# B&R Automation Studio project vibratorControlWithCurrentController (part 2)

### Hardware
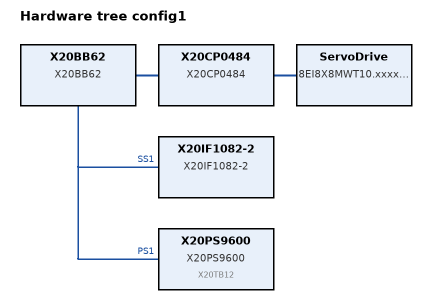
[picture p1: hardware tree config1]
```
ServoDrive : 8EI8X8MWT10.xxxx-1 v2.3.2.0  [PLK1 -> X20CP0484.IF3 (NodeNumber=1) [Cable Type=PowerlinkCable, Length=10, Version=1.0.0.3]]
  MotionTP = Acp10Arnc0
  Ax1Interface = Ax1EnDat
X20BB62 : X20BB62 v1.3.0.0
  Connector IF6:
    CycleTime = 1600
    AsyncPayload = 120
    OutputJustInTime = off
X20CP0484 : X20CP0484 v1.7.0.0  [SL -> X20BB62.SL1]
  Connector IF2:
    ActivateDevice = 1
    HostName = countingmachine
    Mode = Manual
    InternetAddress = 192.168.2.11
    SubnetMask = 255.255.255.0
    InaNodeNumber = 0
    ActivateSnmp = 2
  Connector IF3:
    MtuSize = 1500
    CycleTime = 800
    InternetAddress = 192.168.200.240
    SubnetMask = 255.255.255.0
    ActivateANSL = 1
  ConfigurationID = vibratorControlWithCurrentController
  UserPartitionSize = 100
  RemanentGlobalPvSize = 500
  VolatileGlobalPvSize = 455350
  EnableUsbRemoteInstall = 1
  EnableCfRemoteInstall = 1
  TimerDeviceType = EPLX2X
  TimerDevice = X20CP0484.IF3
  IdleTaskClass = 4
  TaskClassIdleTime = 1600
  CyclicTaskClassCount = 5
  Cyclic1Duration = 800
  Cyclic1Tolerance = 0
  Cyclic2Duration = 1600
  Cyclic2Tolerance = 0
  Cyclic3Duration = 4800
  Cyclic3Tolerance = 0
  Cyclic4Duration = 20000
  Cyclic4Tolerance = 1000000
  Cyclic5Duration = 40000
  Cyclic5Tolerance = 1000000
  Cyclic6Duration = 500000
  Cyclic6Tolerance = 500000
  Cyclic7Duration = 1000000
  Cyclic7Tolerance = 1000000
  Cyclic8Duration = 9600
  Cyclic8Tolerance = 30000000
  FileDevice1
  FileDeviceName1 = USER
  FileDevicePath1 = USER_PATH
  TimeZone = 140
  ActivateSntp = 1
  SntpcServAddr1 = 192.168.1.199
  EthernetHostName = cm20
  EthernetDefaultGateway = 192.168.1.254
  ActivateDns = 1
  DnsServer1 = 192.168.1.1
  FtpUser1
  FtpUsername1 = admin
  FtpUserPassword1 = /xeWp7dP4cZARaoRUYb4lC4ZD6ydIPKFJHxZK63t4D4=
  FtpUserSalt1 = z+XtgaLv
  FTPAccessRight1 = 0
  FtpUser2
  FtpUsername2 = superuser
  FtpUserPassword2 = hun78AKmVJbSvtD9VGxdA3Iq+bPiFMAeRRsTULM9hlc=
  FtpUserSalt2 = IDYkuK0C
  FTPAccessRight2 = 0
  FTPdevice2 = ALL
  FtpUser3
  FtpUsername3 = update
  FtpUserPassword3 = +43P0CP5LPvLZS5Hk18lIwvQq9JpaLJM6nsEQnrbHXY=
  FtpUserSalt3 = TaVVG8PK
  FTPAccessRight3 = 0
  FTPMSpath3 = update
  FtpUser4
  FtpUsername4 = updateewu
  FtpUserPassword4 = epKGN9X0JvLfxgCXyMdS0yy+jyVnLXtvgYSXuK2LydA=  // updateewu
  FtpUserSalt4 = ShQX0Ew+
  FTPAccessRight4 = 0
  FTPMSpath4 = updateewu
  ActivateOpcUa = 1
  OpcUaInformationModels_PV_Version = 2
  OpcUaInformationModel_Facet = 0
  OpcUaInformationModel_TypeInformation = 0
  OpcUaInformationModel_BaseObjectTypeForStructures = 0
X20IF1082-2 : X20IF1082-2 v1.15.0.0  [SS -> X20BB62.SS1]
  Connector IF1:
    Operation = EthOnly
    HostName = cm20
    ActivateANSL = 1
    ActivateSnmp = 2
X20PS9600 : X20PS9600 v1.6.1.0  [PS -> X20BB62.PS1; SS1 -> X20TB12.SS]
X20TB12 : X20TB12 v1.0.0.0
```

### Acp10map.ncm - X20CP0484/Motion/Acp10map.ncm
```
NcMapping (NcSwId=Acp10, DisabledNodesAreHidden=False)
  NcObject gAxisBelt (ModuleId=ServoDrive, Type=ncAXIS, Channel=1, AcoposSimulation=Off, InitParameter=gAxisBelti, AcoposParameter=gAxisBelta, Disabled=TRUE, ModuleDisabled=FALSE)
  NcObject gAxisVibL (ModuleId=ServoDrive, Type=ncAXIS, Channel=2, AcoposSimulation=Off, InitParameter=gAxisVibLi, AcoposParameter=lfNew, Disabled=TRUE, ModuleDisabled=FALSE)
  NcObject 8EI8X8MWT10.xxxx-1_ncV_AXIS1 (ModuleId=ServoDrive, Type=ncV_AXIS, Channel=1, Disabled=TRUE, ModuleDisabled=FALSE)
  NcObject 8EI8X8MWT10.xxxx-1_ncV_AXIS2 (ModuleId=ServoDrive, Type=ncV_AXIS, Channel=2, Disabled=TRUE, ModuleDisabled=FALSE)
  NcObject gAxisVibC (ModuleId=ServoDrive, Type=ncAXIS, Channel=3, AcoposSimulation=Off, InitParameter=gAxisVibCi, AcoposParameter=cfCurCtr, Disabled=FALSE, ModuleDisabled=FALSE)
  NcObject ServoDrive_ncV_AXIS3 (ModuleId=ServoDrive, Type=ncV_AXIS, Channel=3, AcoposSimulation=off, Disabled=true, ModuleDisabled=FALSE)
```

## Logical view

Binary libraries used (declarations not repeated): operator, runtime, astime, AsIecCon, Acp10man, Acp10par, NcGlobal, MpRecipe, MpBase, sys_lib, MpAlarmX, Acp10_MC, AsBrMath, standard, AsBrStr, brsystem, DataObj, AsOpcUas, ArProject, AsSem, AsIO, AsOpcUac, FileIO, AsIODiag, AsUSB, RandomLib, AsHttp, AsARCfg, AsMath, asstring, AsEthIP, MTTypes, MpData, MpServer, EasyUaClnt, AsIOLink, AsIOAcc, AsUDP, MTData, MTBasics, MTFilter, MTLookUp 5.24.1, MpReport 5.23.1

### Global.typ - Global data types
```iecst
TYPE
	copy_recipe_command_typ :
		(
		COPY_RECIPE_NONE := 0,
		COPY_RECIPE_NEXT_TO_WORKING := 1,
		COPY_RECIPE_SANDBOX_TO_NEXT := 2
		);
END_TYPE
```

### Global.var - Global variables
```iecst
VAR
	gMachineType : STRING[10];
END_VAR
VAR CONSTANT
	MODE_EMPTY : DINT := 21;
	MODE_TEACH_CAPCON : DINT := 25;
	MODE_TEACH_BELT : DINT := 26;
END_VAR
VAR
	gAxisVibC : ACP10AXIS_typ;
	gAxisVibL : ACP10AXIS_typ;
	gAxisBelt : ACP10AXIS_typ;
END_VAR
```

### Package Logical/Libraries - Global libraries

### Library Logical/Libraries/brdkMC (IEC, version 2.02.2) - Basic motion library
Depends on: Runtime, Acp10_MC, AsBrMath, standard, AsBrStr

#### brdkMC.typ - Exported data types
```iecst
TYPE
	brdk_mc_para_hwinputs_typ : 	STRUCT  (*HW inputs*)
		homeReference : brdk_mc_para_hwinputs_di_typ; (*Home switch*)
		negHwLimit : brdk_mc_para_hwinputs_di_typ; (*Negative hw limit switch*)
		posHwLimit : brdk_mc_para_hwinputs_di_typ; (*Positive hw limit switch*)
		trigger1 : brdk_mc_para_hwinputs_di_typ; (*Trigger switch*)
		trigger2 : brdk_mc_para_hwinputs_di_typ; (*Trigger switch*)
	END_STRUCT;
	brdk_mc_para_hwinputs_di_typ : 	STRUCT  (*HW input commands*)
		input : BOOL; (*Manipulates switch in the drive if useExternalInput is TRUE*)
		useExternalInput : BOOL; (*Get the input from a digital input module or PLC*)
	END_STRUCT;
	brdk_mc_command_typ : 	STRUCT  (*Commands*)
		power : BOOL; (*Power on drive*)
		home : BOOL; (*Home axis*)
		moveAbsolute : BOOL; (*Move to position*)
		moveAdditive : BOOL; (*Move distance*)
		moveVelocity : BOOL; (*Move with speed*)
		halt : BOOL; (*Halt movement*)
		stop : BOOL; (*Stop movement*)
		jogPositive : BOOL; (*Jog in positive direction*)
		jogNegative : BOOL; (*Jog in negative direction*)
		gearIn : BOOL; (*Connect slave axis to master axis*)
		gearOut : BOOL; (*Disconnect master and slave axes*)
		limitLoad : BOOL; (*Limits the motor torque*)
		errorAcknowledge : BOOL; (*Acknowledge error at rising edge*)
		updatePeriod : BOOL; (*Update axis factor and period, done automatically at axis bootup*)
		simulateError : BOOL; (*Trigger a simulated axis error*)
		resetTorqueStatus : BOOL; (*Reset torque statistics*)
		newBatAcknowledge : BOOL; (*Acknowledge battery excange - Only for AcoposMicro with Endat 2.2*)
	END_STRUCT;
	brdk_mc_status_typ : 	STRUCT  (*Status*)
		state : Status_enum; (*Current PLCopen state*)
		actVelocity : REAL; (*Actual velocity [PLCopen units/s]*)
		actPosition : REAL; (*Actual position [PLCopen units]*)
		actLagError : REAL; (*Actual position lag error [PLCopen units] if configuration factor set > 0 else in [units]*)
		actTorque : REAL; (*Actual torque [Nm]*)
		torque : brdk_mc_status_torque_typ; (*Extended torque readout*)
		powerOn : BOOL; (*Axis is powered on*)
		isHomed : BOOL; (*Axis is homed*)
		inMotion : BOOL; (*Axis is in motion or geared in to a master axis*)
		stopped : BOOL; (*Axis is stopped using the command stop and is at standstill*)
		done : BOOL; (*Specified command done*)
		busy : BOOL; (*Specified command is executed and active*)
		updateDone : BOOL; (*UpdatePeriod command done*)
		error : brdk_mc_status_error_typ; (*Error status information*)
		driveStatus : brdk_mc_status_drive_status_typ; (*Drive status information*)
		encoderBatteryStatus : brdk_mc_enc_bat_status_typ; (*Status of encoder battery - Only for AcoposMicro with Endat 2.2*)
		axisDescription : STRING[30]; (*Defined axis desciption*)
	END_STRUCT;
	brdk_mc_status_drive_status_typ : 	STRUCT  (*Drive status*)
		simulation : BOOL; (*If TRUE, simulation mode is active for the drive.*)
		initialized : BOOL; (*If TRUE, the network is initialized.*)
		homeSwitch : BOOL; (*If TRUE, the digital reference switch input is active.*)
		posLimitSwitch : BOOL; (*If TRUE, the positive hardware limit switch is active.*)
		negLimitSwitch : BOOL; (*If TRUE, the negative hardware limit switch is active.*)
		trigger1 : BOOL; (*If TRUE, the first trigger input is active.*)
		trigger2 : BOOL; (*If TRUE, the second trigger input is active.*)
		driveEnable : BOOL; (*If TRUE, the enable input is in use.*)
		controllerReady : BOOL; (*If TRUE, the controller is ready to be turned on.*)
		lagWarning : BOOL; (*If TRUE, the lag error has exceeded the limit value specified for a warning (limit.parameter.ds_warning).*)
	END_STRUCT;
	brdk_mc_status_error_text_typ : 	STRUCT  (*Error text*)
		active : ARRAY[0..4]OF STRING[363]; (*Active fault descriptions*)
		last : ARRAY[0..4]OF STRING[363]; (*Last reset faults descriptions*)
	END_STRUCT;
	brdk_mc_status_error_typ : 	STRUCT  (*Error status*)
		fault : BOOL; (*Fault present on axis*)
		count : UINT; (*Number of faults*)
		text : brdk_mc_status_error_text_typ; (*Error message*)
	END_STRUCT;
	brdk_mc_status_torque_typ : 	STRUCT  (*Torque status*)
		actual : REAL; (*Actual torque 0.5 sec average [Nm]*)
		continous : REAL; (*Continous peak torque 5 sec average [Nm]*)
		peak : REAL; (*Peak torque 0.5 sec average [Nm]*)
	END_STRUCT;
	brdk_mc_internal_typ : 	STRUCT  (*internal*)
		MC_BR_CyclicRead_1 : MC_BR_CyclicRead;
		MC_MoveVelocity_0 : MC_MoveVelocity;
		MC_Reset_0 : MC_Reset;
		MC_Home_0 : MC_Home;
		MC_Halt_0 : MC_Halt;
		MC_Stop_0 : MC_Stop;
		MC_Power_0 : MC_Power;
		MC_BR_Simulation_0 : MC_BR_Simulation;
		MC_ReadActualPosition_0 : MC_ReadActualPosition;
		MC_ReadStatus_0 : MC_ReadStatus;
		MC_ReadActualVelocity_0 : MC_ReadActualVelocity;
		MC_GearIn_0 : MC_GearIn;
		MC_GearOut_0 : MC_GearOut;
		MC_MoveAdditive_0 : MC_MoveAdditive;
		MC_MoveAbsolute_0 : MC_MoveAbsolute;
		MC_ReadActualTorque_0 : MC_ReadActualTorque;
		MC_BR_ReadDriveStatus_0 : MC_BR_ReadDriveStatus;
		MC_BR_ReadAxisError_0 : MC_BR_ReadAxisError;
		MC_BR_AxisErrorCollector_0 : MC_BR_AxisErrorCollector;
		MC_BR_GetHardwareInfo_0 : MC_BR_GetHardwareInfo;
		MC_BR_SetHardwareInputs_0 : MC_BR_SetHardwareInputs;
		MC_BR_InitAxisSubjectPar_0 : MC_BR_InitAxisSubjectPar;
		MC_BR_CyclicRead_0 : MC_BR_CyclicRead;
		MC_BR_ReadParID_3 : MC_BR_ReadParID;
		MC_BR_ReadParID_2 : MC_BR_ReadParID;
		MC_BR_ReadParID_1 : MC_BR_ReadParID;
		MC_BR_ReadParID_0 : MC_BR_ReadParID;
		MC_BR_InitModPos_0 : MC_BR_InitModPos;
		MC_BR_CommandError_0 : MC_BR_CommandError;
		MC_BR_WriteParID_1 : MC_BR_WriteParID;
		MC_BR_WriteParID_0 : MC_BR_WriteParID;
		MC_LimitLoad_0 : MC_LimitLoad;
		encoderReset : UDINT;
		old_hardwareInput : brdk_mc_para_hwinputs_typ;
		encoderStatus : UDINT;
		encoderType : USINT;
		strcat_adr : UDINT;
		string2 : STRING[8];
		tmpErrorString : STRING[324];
		tmpErrorCount : UINT;
		tmpErrorID : STRING[5];
		tmpErrorArray : ARRAY[0..3]OF STRING[80];
		i : USINT;
		oldParID : UINT;
		oldErrorID : UINT;
		substate : USINT;
		tmpNumberOfErrors : UINT;
		filterBase : ARRAY[0..1]OF REAL;
		RTInfo : RTInfo;
		calcActualValueTemp_old : REAL;
		calcActualValueTemp : REAL;
		calcActualValue_old : ARRAY[0..1]OF REAL;
		calcActualValue : ARRAY[0..1]OF REAL;
		filterTime : ARRAY[0..1]OF REAL;
		stateMotor : USINT;
		filterBaseTemp : REAL;
		filterTimeTemp : REAL;
		TON_error_read_delay : TON;
		k : USINT;
		batteryState : bat_state_enum;
		acoposMicroBatMon : BOOL;
		tmpDriveStatus : MC_DRIVESTATUS_TYP;
		initialized : BOOL;
	END_STRUCT;
	brdk_mc_parameter_typ : 	STRUCT  (*Parameters*)
		position : REAL; (*Position for an absolute movement [PLCopen units]*)
		distance : REAL; (*Distance for an additive movement [PLCopen units]*)
		velocity : REAL; (*Movement velocity [PLCopen units/s] *)
		acceleration : REAL; (*Acceleration [PLCopen units/s²]*)
		deceleration : REAL; (*Deceleration [PLCopen units/s²]*)
		decelerationFault : REAL; (*Deceleration at axis fault [PLCopen units/s²]*)
		direction : USINT; (*Movement direction:
mcPOSITITVE_DIR ... 0

mcNEGATIVE_DIR ... 1

mcCURRENT_DIR ... 2

mcSHORTEST_WAY ... 3

mcEXCEED_PERIOD ... 8*)
		loadLimit : REAL; (*Torque load limit [Nm]*)
		homePosition : REAL; (*Home position, position after homing [PLCopen units]*)
		homeMode : USINT; (*Homing mode:
mcHOME_ABS_SWITCH (performs homing with absolute reference switch)

mcHOME_SWITCH_GATE (homing with reference switch gate)

mcHOME_LIMIT_SWITCH (homing with hardware limit switch)

mcHOME_DIRECT (direct homing without reference pulse)

mcHOME_REF_PULSE (direct homing with reference pulse)

mcHOME_ABSOLUTE (homing by setting the homing offset)

mcHOME_ABSOLUTE_CORR (homing by setting the homing offset with counting range correction)

mcHOME_DCM (homing using interval-encoded reference marks)

mcHOME_DCM_CORR (Homing using distance coded reference marks with counting range correction)

mcHOME_RESTORE_POS (restore position from permanent memory)

mcHOME_AXIS_REF (performs homing with the data from the axis structure)

mcHOME_BLOCK_TORQUE (performs homing to mechanical limit, torque as criteria)

mcHOME_BLOCK_DS (performs homing to mechanical limit, lag error value as criteria)*)
		ratioSlave : INT; (*Slave gear ratio*)
		ratioMaster : UINT; (*Master gear ration*)
		gearInMasterParID : UINT; (*This ParID is used instead of the position setpoint;
0 ... Use position setpoint*)
		gearInMasterParIDMaxVelocity : REAL; (*If this parameter is "0.0", the current velocity of the master axis is used.
If a value is specified for "MasterParID":
Maximum velocity of the master ParID value

If a value is not specified for "MasterParID":
Maximum velocity of the master axis [PLCopen units of master/s]*)
		errorSimulationCommand : USINT; (*0: Warning message reported

1: Error message reported

2: Error message reported and active movement aborted

3: Error message reported, active movement aborted and controller switched off

4: Error message reported, active movement ended with a speed-controlled ramp and controller switched off*)
		hwInput : brdk_mc_para_hwinputs_typ; (*Hardware input manipulation for home reference, triggers and limit switches*)
	END_STRUCT;
	brdk_mc_configuration_typ : 	STRUCT  (*Axis configuration*)
		masterAxis : UDINT; (*Master axis reference*)
		axis : UDINT; (*Axis reference*)
		errorTextObject : STRING[12]; (*Name of the acp10 error text object
If no name is entered, the default name 'acp10etxen' is assumed (table must be available in the project)*)
		description : STRING[30]; (*Optional: Axis description or name; added to the error texts*)
		factor : UDINT; (*Axis factor*)
		period : UDINT; (*Axis period*)
		ignoreSwLimit : USINT; (*Ignore software end limit positions (0: end limits active 1: ignore sw end limits)*)
		disableVelocityReading : BOOL; (*Disables actual velocity status readout*)
		disablePositionReading : BOOL; (*Disables actual position status readout*)
		disableTorqueReading : BOOL; (*Disables actual torque status readout*)
		disableTemperatureReading : BOOL; (*Disables actual motor temperature readout*)
		disableLagErrorReading : BOOL; (*Disables actual lag error status readout*)
	END_STRUCT;
	brdk_mc_info_typ : 	STRUCT  (*HW info*)
		startupPhase : STRING[100]; (*Drive startup phase information*)
		hw : brdk_mc_info_hw_typ; (*Hardware information*)
	END_STRUCT;
	brdk_mc_info_hw_typ : 	STRUCT  (*Hardware information*)
		drive : brdk_mc_info_hw_drive_typ; (*Motor type*)
		motor : brdk_mc_info_hw_motor_typ; (*Motors maximum torque [Nm]*)
	END_STRUCT;
	brdk_mc_info_hw_drive_typ : 	STRUCT  (*HW drive info*)
		model : STRING[32]; (*Drive model number*)
		serial : STRING[32]; (*Drive serial number*)
		card : ARRAY[0..3]OF brdk_mc_info_hw_card_typ; (*Plugin cards*)
	END_STRUCT;
	brdk_mc_info_hw_card_typ : 	STRUCT  (*HW card info*)
		model : STRING[32]; (*Model number*)
		serial : STRING[32]; (*Serial number*)
	END_STRUCT;
	brdk_mc_info_hw_motor_typ : 	STRUCT  (*Motor info*)
		model : STRING[32]; (*Motor type*)
		temperature : REAL; (*Motor temperature [C]*)
		torqueRated : REAL; (*Motors nominal torque [Nm]*)
		torqueMaximum : REAL; (*Motors maximum torque [Nm]*)
	END_STRUCT;
	brdk_mc_enc_bat_status_typ : 	STRUCT  (*Encoder battry information*)
		batteryOK : BOOL; (*Encoder battery is OK - Voltage OK and position valid*)
		batteryError : BOOL; (*Encoder battery NOT ok - voltage has dropped below threshhold. Posiion valid if PositionLost = false.*)
		batteryWarning : BOOL; (*Error has been acknowledged - battery not exchanged, position still valid*)
		positionLost : BOOL; (*Encoder postion has been lost due to battery failure*)
	END_STRUCT;
	state_enum :
		(
		ST_INIT := 0,
		ST_WAIT := 1,
		ST_POWER_ON := 2,
		ST_HOME_AT_POWER_OFF := 3,
		ST_EXTERNAL_HW_INPUTS := 5,
		ST_UPDATE_FACTOR_PERIOD := 6,
		ST_READY := 10,
		ST_HOME := 20,
		ST_STOP := 30,
		ST_HALT := 31,
		ST_MOVE_ABSOLUTE := 40,
		ST_MOVE_ADDITIVE := 41,
		ST_MOVE_VELOCITY := 42,
		ST_GEAR_START := 50,
		ST_GEAR_STOP := 51,
		ST_IN_GEAR := 52,
		ST_JOG_POS := 60,
		ST_JOG_NEG := 61,
		ST_HALT_JOG := 62,
		ST_STOP_AFTER_ERROR := 100,
		ST_STOPPING_AFTER_ERROR := 101,
		ST_ERROR := 110,
		ST_CHECK_ERROR := 111,
		ST_ERROR_RESET := 120,
		ST_ENCODER_ERROR_RESET := 130
		);
	bat_state_enum :
		(
		ST_BAT_OK := 0,
		ST_BAT_ERROR := 1,
		ST_BAT_WARNING := 2,
		ST_BAT_POS_LOST := 3
		);
	Status_enum :
		(
		DISABLED := 0,
		STANDSTILL := 1,
		HOMING := 2,
		CONTINOUS_MOTION := 3,
		DISCRETE_MOTION := 4,
		SYNCHRONIZED_MOTION := 5,
		STOPPING := 6,
		ERROR_STOP := 10
		);
END_TYPE
```

#### brdkMC.fun - Exported functions and function blocks
```iecst
FUNCTION_BLOCK brdkMcBasic (*brdk Motion basic*)
	VAR_INPUT
		command : brdk_mc_command_typ; (*command input*)
		parameter : brdk_mc_parameter_typ; (*parameter input*)
		configuration : brdk_mc_configuration_typ; (*configuration input*)
	END_VAR
	VAR_OUTPUT
		status : brdk_mc_status_typ; (*status output*)
		info : brdk_mc_info_typ; (*information output*)
	END_VAR
	VAR
		state : state_enum; (*state enumeration*)
		internal : brdk_mc_internal_typ; (*internal structure*)
		pAxis : REFERENCE TO ACP10AXIS_typ; (*internal axis pointer reference*)
	END_VAR
END_FUNCTION_BLOCK

FUNCTION dstoa : UINT (****)
	VAR_INPUT
		driveState : Status_enum;
		pString : UDINT;
	END_VAR
END_FUNCTION
```

#### brdkMcBasic.st
```iecst
FUNCTION_BLOCK  brdkMcBasic

	(* Access the axis structure *)
	pAxis ACCESS configuration.axis;

	(*********************** CHECK FOR ERRORS **************************)
	IF (state < ST_STOP_AFTER_ERROR) THEN
		IF (internal.MC_BR_AxisErrorCollector_0.Errorstop) THEN
			state := ST_ERROR;
		ELSIF (internal.MC_BR_AxisErrorCollector_0.FunctionBlockError) OR
		   	  (internal.MC_BR_AxisErrorCollector_0.AxisError) OR
			  (internal.MC_BR_AxisErrorCollector_0.AxisWarning) THEN
			status.busy := 0;
			status.done := 0;
			state 		:= ST_STOP_AFTER_ERROR;
		END_IF
	END_IF

	(***************** CHECK IF POWER SHOULD BE OFF *******************)
	IF (command.power = 0 AND state < ST_STOP_AFTER_ERROR AND state <> ST_HOME_AT_POWER_OFF AND state <> ST_INIT AND state <> ST_EXTERNAL_HW_INPUTS AND state <> ST_UPDATE_FACTOR_PERIOD) THEN
		status.busy := 0;
		status.done := 0;

		IF ((internal.MC_ReadStatus_0.Errorstop = 1) AND (internal.MC_ReadStatus_0.Valid = TRUE)) THEN
			state := ST_ERROR_RESET;
		ELSE
			state := ST_WAIT;
		END_IF
	END_IF

	(* Status Motion States *)
	IF internal.MC_ReadStatus_0.Disabled THEN
		status.state := DISABLED;
	ELSIF internal.MC_ReadStatus_0.StandStill THEN
		status.state := STANDSTILL;
	ELSIF internal.MC_ReadStatus_0.Homing THEN
		status.state := HOMING;
	ELSIF internal.MC_ReadStatus_0.Stopping THEN
		status.state := STOPPING;
	ELSIF internal.MC_ReadStatus_0.Errorstop THEN
		status.state := ERROR_STOP;
	ELSIF internal.MC_ReadStatus_0.DiscreteMotion THEN
		status.state := DISCRETE_MOTION;
	ELSIF internal.MC_ReadStatus_0.ContinuousMotion THEN
		status.state := CONTINOUS_MOTION;
	ELSIF internal.MC_ReadStatus_0.SynchronizedMotion THEN
		status.state := SYNCHRONIZED_MOTION;
	END_IF

	(* Limit load torque *)
	internal.MC_LimitLoad_0.Load		:= parameter.loadLimit;
	internal.MC_LimitLoad_0.Direction	:= parameter.direction;
	internal.MC_LimitLoad_0.Enable		:= command.limitLoad;

	(***************************************************************)
	(************************* MAIN CONTROL ************************)
	(***************************************************************)

	(* check for stop command *)
	IF command.stop AND state <> ST_INIT AND state <> ST_WAIT AND state <> ST_POWER_ON AND state <> ST_UPDATE_FACTOR_PERIOD AND state <> ST_HOME_AT_POWER_OFF AND state <> ST_EXTERNAL_HW_INPUTS AND state <> ST_STOP AND state < 100 THEN
		internal.MC_Stop_0.Deceleration	:= parameter.deceleration;
		internal.MC_Stop_0.Execute 		:= 1;
		state := ST_STOP;
	END_IF

	CASE state OF

		(****************** STARTING DRIVE *****************)
		ST_INIT:
			CASE internal.substate OF
				0:
					IF pAxis.network.phase = 90 THEN
						internal.substate := 10;
					END_IF

				10:	(* initialize factor and period *)
					internal.MC_BR_InitModPos_0.Factor	:= configuration.factor;
					internal.MC_BR_InitModPos_0.Period	:= configuration.period;
					internal.MC_BR_InitModPos_0.Execute	:= TRUE;

					IF internal.MC_BR_InitModPos_0.Done THEN
						internal.MC_BR_InitModPos_0.Execute := FALSE;
						internal.substate					:= 20;
					END_IF

				20: (* set end limit ignore *)
					internal.MC_BR_WriteParID_1.ParID		:= ACP10PAR_SGEN_SW_END_IGNORE;
					internal.MC_BR_WriteParID_1.DataType	:= ncPAR_TYP_USINT;
					internal.MC_BR_WriteParID_1.DataAddress	:= ADR(configuration.ignoreSwLimit);
					internal.MC_BR_WriteParID_1.Execute		:= TRUE;

					IF internal.MC_BR_WriteParID_1.Done THEN
						internal.MC_BR_WriteParID_1.Execute := FALSE;
						internal.initialized				:= TRUE;
						internal.substate 					:= 0;
						state 								:= ST_WAIT;
					END_IF
					internal.MC_BR_WriteParID_1(Axis := configuration.axis);
			END_CASE

		(******************** WAIT *************************)
		ST_WAIT: (* STATE: Wait *)

			(* reset status *)
			status.busy   		:= 0;
			status.done 		:= 0;
			status.updateDone 	:= 0;

			(* reset user commands *)
			command.stop 			:= 0;
			command.halt 			:= 0;
			command.moveVelocity	:= 0;
			command.moveAbsolute	:= 0;
			command.moveAdditive	:= 0;
			command.gearIn 			:= 0;
			command.gearOut			:= 0;
			command.jogPositive		:= 0;
			command.jogNegative		:= 0;

			(* reset all fb execute inputs we use *)
			internal.MC_Home_0.Execute 					:= 0;
			internal.MC_Stop_0.Execute 					:= 0;
			internal.MC_Halt_0.Execute 					:= 0;
			internal.MC_MoveAbsolute_0.Execute 			:= 0;
			internal.MC_MoveAdditive_0.Execute 			:= 0;
			internal.MC_MoveVelocity_0.Execute 			:= 0;
			internal.MC_GearIn_0.Execute 				:= 0;
			internal.MC_GearOut_0.Execute 				:= 0;
			internal.MC_BR_ReadAxisError_0.Acknowledge	:= 0;
			internal.MC_Reset_0.Execute 				:= 0;
			internal.substate 							:= 0;

			IF (command.power) THEN
				state := ST_POWER_ON;
			ELSE
				internal.MC_Power_0.Enable := 0;
			END_IF

			(* wait for homing command *)
			IF (command.home) THEN
				internal.MC_Home_0.Position 	:= parameter.homePosition;
				internal.MC_Home_0.HomingMode 	:= parameter.homeMode;
				internal.MC_Home_0.Execute 		:= 1;
				state 							:= ST_HOME_AT_POWER_OFF;
			END_IF

			(* initialize factor and period *)
			IF command.updatePeriod THEN
				internal.MC_BR_InitModPos_0.Axis 	:= configuration.axis;
				internal.MC_BR_InitModPos_0.Factor	:= configuration.factor;
				internal.MC_BR_InitModPos_0.Period	:= configuration.period;
				internal.MC_BR_InitModPos_0.Execute	:= TRUE;
				state 								:= ST_UPDATE_FACTOR_PERIOD;
			END_IF

			(* check if external inputs has been changed *)
			IF parameter.hwInput.homeReference.useExternalInput <> internal.old_hardwareInput.homeReference.useExternalInput OR
			   parameter.hwInput.negHwLimit.useExternalInput <> internal.old_hardwareInput.negHwLimit.useExternalInput OR
			   parameter.hwInput.posHwLimit.useExternalInput <> internal.old_hardwareInput.posHwLimit.useExternalInput OR
			   parameter.hwInput.trigger1.useExternalInput <> internal.old_hardwareInput.trigger1.useExternalInput OR
			   parameter.hwInput.trigger2.useExternalInput <> internal.old_hardwareInput.trigger2.useExternalInput THEN
				IF parameter.hwInput.homeReference.useExternalInput <> internal.old_hardwareInput.homeReference.useExternalInput THEN
					IF parameter.hwInput.homeReference.useExternalInput THEN
						pAxis.dig_in.level.reference.5 := pAxis.dig_in.level.reference.8 := 1;
					ELSE
						pAxis.dig_in.level.reference.5 := pAxis.dig_in.level.reference.8 := 0;
					END_IF
				END_IF
				IF parameter.hwInput.negHwLimit.useExternalInput <> internal.old_hardwareInput.negHwLimit.useExternalInput THEN
					IF parameter.hwInput.negHwLimit.useExternalInput THEN
						pAxis.dig_in.level.neg_hw_end.5 := pAxis.dig_in.level.neg_hw_end.8 := 1;
					ELSE
						pAxis.dig_in.level.neg_hw_end.5 := pAxis.dig_in.level.neg_hw_end.8 := 0;
					END_IF
				END_IF
				IF parameter.hwInput.posHwLimit.useExternalInput <> internal.old_hardwareInput.posHwLimit.useExternalInput THEN
					IF parameter.hwInput.posHwLimit.useExternalInput THEN
						pAxis.dig_in.level.pos_hw_end.5 := pAxis.dig_in.level.pos_hw_end.8 := 1;
					ELSE
						pAxis.dig_in.level.pos_hw_end.5 := pAxis.dig_in.level.pos_hw_end.8 := 0;
					END_IF
				END_IF
				IF parameter.hwInput.trigger1.useExternalInput <> internal.old_hardwareInput.trigger1.useExternalInput THEN
					IF parameter.hwInput.trigger1.useExternalInput THEN
						pAxis.dig_in.level.trigger1.5 := pAxis.dig_in.level.trigger1.8 := 1;
					ELSE
						pAxis.dig_in.level.trigger1.5 := pAxis.dig_in.level.trigger1.8 := 0;
					END_IF
				END_IF
				IF parameter.hwInput.trigger2.useExternalInput <> internal.old_hardwareInput.trigger2.useExternalInput THEN
					IF parameter.hwInput.trigger2.useExternalInput THEN
						pAxis.dig_in.level.trigger2.5 := pAxis.dig_in.level.trigger2.8 := 1;
					ELSE
						pAxis.dig_in.level.trigger2.5 := pAxis.dig_in.level.trigger2.8 := 0;
					END_IF
				END_IF

				internal.old_hardwareInput.homeReference.useExternalInput 	:= parameter.hwInput.homeReference.useExternalInput;
				internal.old_hardwareInput.negHwLimit.useExternalInput 		:= parameter.hwInput.negHwLimit.useExternalInput;
				internal.old_hardwareInput.posHwLimit.useExternalInput 		:= parameter.hwInput.posHwLimit.useExternalInput;
				internal.old_hardwareInput.trigger1.useExternalInput 		:= parameter.hwInput.trigger1.useExternalInput;
				internal.old_hardwareInput.trigger2.useExternalInput 		:= parameter.hwInput.trigger2.useExternalInput;
				state 														:= ST_EXTERNAL_HW_INPUTS;
			END_IF

			(* check if drive was initialized *)
			IF NOT internal.initialized	THEN
				internal.substate := 0;
				state 			  := ST_INIT;
			END_IF

		(******************** POWER ON **********************)
		ST_POWER_ON: (* STATE: Power on *)
			internal.MC_Power_0.Enable := 1;
			IF (internal.MC_Power_0.Status = 1) THEN
				state := ST_READY;
			END_IF

			(* check if error occured *)
			IF (internal.MC_Power_0.Error) THEN
				internal.MC_Power_0.Enable := 0;
				state := ST_WAIT;
			END_IF

		(******************** HOME AT POWER OFF *************)
		ST_HOME_AT_POWER_OFF: (* STATE: start homing process *)
			(* check if functionblock is busy *)
			status.busy := internal.MC_Home_0.Busy;

			(* if axis homed go to state ready *)
			status.done := internal.MC_Home_0.Done;

			(* return to ready state *)
			IF NOT command.home THEN
				status.busy := 0;
				status.done := 0;
				internal.MC_Home_0.Execute := 0;
				state := ST_WAIT;
			END_IF

		(********* setup EXTERNAL HW INPUTS **************)
		ST_EXTERNAL_HW_INPUTS:
			(* check if functionblock is busy *)
			status.busy := internal.MC_BR_InitAxisSubjectPar_0.Busy;

			(* check if command is done *)
			status.done := internal.MC_BR_InitAxisSubjectPar_0.Done;

			internal.MC_BR_InitAxisSubjectPar_0.Execute := TRUE;

			IF internal.MC_BR_InitAxisSubjectPar_0.Done THEN
				internal.MC_BR_InitAxisSubjectPar_0.Execute := FALSE;
				state 										:= ST_WAIT;
			END_IF

		(********* UPDATE period AND factor **************)
		ST_UPDATE_FACTOR_PERIOD:
			status.updateDone := internal.MC_BR_InitModPos_0.Done AND internal.MC_BR_WriteParID_1.Done;

			IF internal.MC_BR_InitModPos_0.Done THEN
				internal.MC_BR_WriteParID_1.ParID		:= ACP10PAR_SGEN_SW_END_IGNORE;
				internal.MC_BR_WriteParID_1.DataType	:= ncPAR_TYP_USINT;
				internal.MC_BR_WriteParID_1.DataAddress	:= ADR(configuration.ignoreSwLimit);
				internal.MC_BR_WriteParID_1.Execute		:= TRUE;
			END_IF

			IF NOT command.updatePeriod THEN
				internal.MC_BR_WriteParID_1.Execute	:= FALSE;
				internal.MC_BR_InitModPos_0.Execute := FALSE;
				state 	 							:= ST_WAIT;
			END_IF

		(******************** READY **********************)
		ST_READY: (* STATE: Waiting for commands *)
			IF command.home AND NOT internal.MC_Home_0.CommandAborted THEN
				internal.MC_Home_0.Position 	:= parameter.homePosition;
				internal.MC_Home_0.HomingMode 	:= parameter.homeMode;
				state := ST_HOME;

			ELSIF command.halt AND NOT internal.MC_Halt_0.CommandAborted THEN
				internal.MC_Halt_0.Deceleration	:= parameter.deceleration;
				state := ST_HALT;

			ELSIF command.moveAbsolute AND NOT internal.MC_MoveAbsolute_0.CommandAborted THEN
				internal.MC_MoveAbsolute_0.Position		:= parameter.position;
				internal.MC_MoveAbsolute_0.Velocity		:= parameter.velocity;
				internal.MC_MoveAbsolute_0.Acceleration	:= parameter.acceleration;
				internal.MC_MoveAbsolute_0.Deceleration	:= parameter.deceleration;
				internal.MC_MoveAbsolute_0.Direction	:= parameter.direction;
				state := ST_MOVE_ABSOLUTE;

			ELSIF command.moveAdditive AND NOT internal.MC_MoveAdditive_0.CommandAborted THEN
				internal.MC_MoveAdditive_0.Distance		:= parameter.distance;
				internal.MC_MoveAdditive_0.Velocity		:= parameter.velocity;
				internal.MC_MoveAdditive_0.Acceleration	:= parameter.acceleration;
				internal.MC_MoveAdditive_0.Deceleration	:= parameter.deceleration;
				state := ST_MOVE_ADDITIVE;

			ELSIF command.moveVelocity AND NOT internal.MC_MoveVelocity_0.CommandAborted THEN
				internal.MC_MoveVelocity_0.Velocity		:= parameter.velocity;
				internal.MC_MoveVelocity_0.Acceleration	:= parameter.acceleration;
				internal.MC_MoveVelocity_0.Deceleration	:= parameter.deceleration;
				internal.MC_MoveVelocity_0.Direction	:= parameter.direction;
				state := ST_MOVE_VELOCITY;

			ELSIF command.jogPositive AND NOT internal.MC_MoveVelocity_0.CommandAborted THEN
				internal.MC_MoveVelocity_0.Velocity		:= parameter.velocity;
				internal.MC_MoveVelocity_0.Acceleration	:= parameter.acceleration;
				internal.MC_MoveVelocity_0.Deceleration	:= parameter.deceleration;
				internal.MC_MoveVelocity_0.Direction	:= mcPOSITIVE_DIR;
				state := ST_JOG_POS;

			ELSIF command.jogNegative AND NOT internal.MC_MoveVelocity_0.CommandAborted THEN
				internal.MC_MoveVelocity_0.Velocity		:= parameter.velocity;
				internal.MC_MoveVelocity_0.Acceleration	:= parameter.acceleration;
				internal.MC_MoveVelocity_0.Deceleration	:= parameter.deceleration;
				internal.MC_MoveVelocity_0.Direction	:= mcNEGATIVE_DIR;
				state := ST_JOG_NEG;

			ELSIF command.gearIn AND NOT internal.MC_GearIn_0.CommandAborted THEN
				internal.MC_GearIn_0.RatioNumerator			:= parameter.ratioSlave;
				internal.MC_GearIn_0.RatioDenominator		:= parameter.ratioMaster;
				internal.MC_GearIn_0.Acceleration			:= parameter.acceleration;
				internal.MC_GearIn_0.Deceleration			:= parameter.deceleration;
				internal.MC_GearIn_0.MasterParID 			:= parameter.gearInMasterParID;
				internal.MC_GearIn_0.MasterParIDMaxVelocity := parameter.gearInMasterParIDMaxVelocity;
				state := ST_GEAR_START;
			ELSIF command.gearOut THEN
			 	state := ST_GEAR_STOP;
			END_IF

			status.busy	:= 0;
			status.done := 0;

			internal.MC_Home_0.Execute			:= command.home;
			internal.MC_Halt_0.Execute			:= command.halt;
			internal.MC_MoveVelocity_0.Execute  := command.moveVelocity OR command.jogPositive OR command.jogNegative;
			internal.MC_MoveAbsolute_0.Execute 	:= command.moveAbsolute;
			internal.MC_MoveAdditive_0.Execute 	:= command.moveAdditive;
			internal.MC_GearIn_0.Execute 		:= command.gearIn;
			internal.MC_GearOut_0.Execute 		:= command.gearOut;

		(******************** HOME **********************)
		ST_HOME: (* STATE: start homing process *)
			(* check if functionblock is busy *)
			status.busy := internal.MC_Home_0.Busy;

			(* if axis homed go to state ready *)
			status.done := internal.MC_Home_0.Done;

			(* return to ready state *)
			IF NOT command.home THEN
				status.busy := 0;
				status.done := 0;
				internal.MC_Home_0.Execute := 0;
				state := ST_READY;
			END_IF

		(*********************** STOP MOVEMENT *************************)
		ST_STOP: (* STATE: Stop movement *)
			(* check if commanded position is reached *)
			status.done := 0;

			(* check if functionblock is busy *)
			status.busy := internal.MC_Stop_0.Busy;

			(* return to ready state *)
			IF NOT command.stop THEN
				status.busy 			:= 0;
				status.done 			:= 0;
				internal.MC_Stop_0.Execute := 0;
				state	 					 := ST_READY;
			END_IF

		(********************** HALT MOVEMENT *************************)
		ST_HALT: (* STATE: Halt movement *)
			(* check if halt is done, velocity zero *)
			status.done := internal.MC_Halt_0.Done;

			(* check if functionblock is busy *)
			status.busy := internal.MC_Halt_0.Busy;

			(* return to ready state *)
			IF NOT command.halt THEN
				status.busy 				:= 0;
				status.done 				:= 0;
				internal.MC_Halt_0.Execute 	:= 0;
				state	 					:= ST_READY;
			END_IF

		(******************** START ABSOLUTE MOVEMENT **********************)
		ST_MOVE_ABSOLUTE: (* STATE: Start absolute movement *)
			(* check if commanded position is reached *)
			status.done := internal.MC_MoveAbsolute_0.Done;

			(* check if functionblock is busy *)
			status.busy := internal.MC_MoveAbsolute_0.Busy;

			(* return to ready state *)
			IF NOT command.moveAbsolute THEN
				status.busy 						:= 0;
				status.done 						:= 0;
				internal.MC_MoveAbsolute_0.Execute  := 0;
				state	 							:= ST_READY;
			END_IF

		(******************** START ADDITIVE MOVEMENT **********************)
		ST_MOVE_ADDITIVE: (* STATE: Start additive movement *)
			(* check if commanded position is reached *)
			status.done := internal.MC_MoveAdditive_0.Done;

			(* check if functionblock is busy *)
			status.busy := internal.MC_MoveAdditive_0.Busy;

			(* return to ready state *)
			IF NOT command.moveAdditive THEN
				status.busy 						:= 0;
				status.done 						:= 0;
				internal.MC_MoveAdditive_0.Execute 	:= 0;
				state	 							:= ST_READY;
			END_IF

		(******************** START VELOCITY MOVEMENT **********************)
		ST_MOVE_VELOCITY: (* STATE: Start velocity movement *)
			(* check if commanded velocity is reached *)
			status.done := internal.MC_MoveVelocity_0.InVelocity;

			(* check if functionblock is busy *)
			status.busy := internal.MC_MoveVelocity_0.Busy;

			(* return to ready state *)
			IF NOT command.moveVelocity THEN
				status.busy 						:= 0;
				status.done 						:= 0;
				internal.MC_MoveVelocity_0.Execute 	:= 0;
				state	 							:= ST_READY;
			END_IF

		(*********************** JOGGING ******************************)
		ST_JOG_POS: (* STATE: Jogging in positive direction *)
			(* check if functionblock is busy *)
			status.busy := internal.MC_MoveVelocity_0.Busy;

			(* return to ready state *)
			IF NOT command.jogPositive THEN
				status.busy 						:= 0;
				status.done 						:= 0;
				internal.MC_MoveVelocity_0.Execute 	:= 0;
				internal.MC_Halt_0.Deceleration		:= parameter.deceleration;
				internal.MC_Halt_0.Execute 			:= 1;
				state	 							:= ST_HALT_JOG;
			END_IF

		(*********************** JOGGING ******************************)
		ST_JOG_NEG: (* STATE: Jogging in positive direction *)
			(* check if functionblock is busy *)
			status.busy := internal.MC_MoveVelocity_0.Busy;

			(* return to ready state *)
			IF NOT command.jogNegative THEN
				status.busy 						:= 0;
				status.done 						:= 0;
				internal.MC_MoveVelocity_0.Execute 	:= 0;
				internal.MC_Halt_0.Deceleration		:= parameter.deceleration;
				internal.MC_Halt_0.Execute 			:= 1;
				state	 							:= ST_HALT_JOG;
			END_IF

		(*********************** JOGGING ******************************)
		ST_HALT_JOG: (* STATE: Stopping jog movement *)
			(* check if functionblock is busy *)
			IF internal.MC_Halt_0.Busy THEN
				internal.MC_Halt_0.Execute := 0;
				state	 				   := ST_READY;
			END_IF

		(******************* START GEAR MOVEMENT **********************)
		ST_GEAR_START: (* STATE: Start electronic gear coupling *)
			(* if axis is in gear go to ready state *)
			status.done := internal.MC_GearIn_0.InGear;

			IF NOT command.gearIn THEN
				status.done 					:= 0;
				internal.MC_GearIn_0.Execute 	:= 0;
				state 							:= ST_READY;
			END_IF

		(******************** STOP GEAR MOVEMENT **********************)
		ST_GEAR_STOP: (* STATE: Stop electronic gear coupling *)
			(* check if coupling is stopped *)
			status.done := internal.MC_GearOut_0.Done;

			IF NOT command.gearOut THEN
				status.done 					:= 0;
				internal.MC_GearOut_0.Execute 	:= 0;
				state 							:= ST_READY;
			END_IF

		(****************** STOP MOVEMENT AFTER ERROR ********************)
		ST_STOP_AFTER_ERROR:
			IF 	(internal.MC_ReadStatus_0.ContinuousMotion) OR
					(internal.MC_ReadStatus_0.DiscreteMotion) OR
					(internal.MC_ReadStatus_0.SynchronizedMotion) OR
					(internal.MC_ReadStatus_0.Homing) THEN

					IF parameter.decelerationFault = 0 THEN
						internal.MC_Stop_0.Deceleration	:= parameter.deceleration;
					ELSE
						internal.MC_Stop_0.Deceleration	:= parameter.decelerationFault;
					END_IF

					status.error.fault 		   := TRUE;
					internal.MC_Stop_0.Execute := 1;
					state					   := ST_STOPPING_AFTER_ERROR;
			ELSE
				state := ST_ERROR;
			END_IF

		(****************** STOPPING MOVEMENT AFTER ERROR ********************)
		ST_STOPPING_AFTER_ERROR:
			(* check if stopped *)
			IF internal.MC_Stop_0.Done THEN
				internal.MC_Stop_0.Execute := 0;
				state	 					 					 := ST_ERROR;
			ELSIF (internal.MC_Stop_0.Error) THEN
				internal.MC_Stop_0.Execute := 0;
				state	 					 					 := ST_ERROR;
			END_IF

			(* check if functionblock is busy *)
			IF internal.MC_Stop_0.Busy THEN
				status.busy := 1;
			END_IF

		(*************** CHECK AND ACKNOWLEDGE ERRORS ********************)
		ST_ERROR:
			(* reset all fb execute inputs we use *)
			IF internal.MC_Power_0.Error OR NOT command.power THEN
 				internal.MC_Power_0.Enable := 0;
			END_IF

			status.busy := 0;
			status.done := 0;

			internal.MC_Home_0.Execute 							:= 0;
			internal.MC_Stop_0.Execute 							:= 0;
			internal.MC_Halt_0.Execute							:= 0;
			internal.MC_MoveAbsolute_0.Execute 					:= 0;
			internal.MC_MoveAdditive_0.Execute 					:= 0;
			internal.MC_MoveVelocity_0.Execute 					:= 0;
			internal.MC_GearIn_0.Execute 						:= 0;
			internal.MC_GearOut_0.Execute 						:= 0;
			internal.MC_BR_ReadAxisError_0.Acknowledge 			:= 0;
			internal.MC_Reset_0.Execute 						:= 0;
			internal.MC_BR_InitModPos_0.Execute					:= 0;

			(* reset user commands *)
			command.stop 				 		:= 0;
			command.halt 		 				:= 0;
			command.home 		 				:= 0;
			command.moveVelocity				:= 0;
			command.moveAbsolute 				:= 0;
			command.moveAdditive 				:= 0;
			command.gearIn 		 				:= 0;
			command.gearOut						:= 0;
			internal.TON_error_read_delay.IN	:= TRUE;

			(* Check for a valid error *)
			IF internal.MC_BR_ReadAxisError_0.Valid AND (internal.MC_BR_ReadAxisError_0.ErrorRecordAvailable OR internal.MC_BR_AxisErrorCollector_0.Errorstop) AND internal.TON_error_read_delay.Q THEN

				(* log error into array *)
				IF internal.tmpErrorCount < SIZEOF(status.error.text.active) / SIZEOF status.error.text.active[0] AND internal.MC_BR_ReadAxisError_0.ErrorRecord.Number <> 0 THEN
					(* add axis description to error text *)
					brsstrcpy(ADR(status.error.text.active[internal.tmpErrorCount]),ADR(configuration.description));
					brsstrcat(ADR(status.error.text.active[internal.tmpErrorCount]), ADR(' - '));

					(* add error id to error text *)
					brsitoa(internal.MC_BR_ReadAxisError_0.ErrorRecord.Number,ADR(internal.tmpErrorID));
					brsstrcat(ADR(status.error.text.active[internal.tmpErrorCount]), ADR(internal.tmpErrorID));
					brsstrcat(ADR(status.error.text.active[internal.tmpErrorCount]),ADR(': '));

					(* add axis error text to error text *)
					internal.tmpErrorString := '';
					FOR internal.i := 0 TO SIZEOF(internal.tmpErrorArray)/SIZEOF(internal.tmpErrorArray[0])-1 DO
						IF brsstrlen(ADR(internal.tmpErrorArray[internal.i])) <> 0 THEN
							brsstrcat(ADR(internal.tmpErrorString),ADR(internal.tmpErrorArray[internal.i]));
							brsstrcat(ADR(internal.tmpErrorString),ADR('. '));
						ELSE
							EXIT;
						END_IF
					END_FOR
					brsstrcat(ADR(status.error.text.active[internal.tmpErrorCount]),ADR(internal.tmpErrorString));
				END_IF

				(* acknowledge axis error *)
				IF (internal.MC_BR_ReadAxisError_0.AxisErrorCount + internal.MC_BR_ReadAxisError_0.AxisWarningCount + internal.MC_BR_ReadAxisError_0.FunctionBlockErrorCount > 0) THEN
					internal.MC_BR_ReadAxisError_0.Acknowledge  := TRUE;
				END_IF

				state := ST_CHECK_ERROR;

			ELSIF internal.MC_BR_ReadAxisError_0.Error AND internal.MC_BR_ReadAxisError_0.ErrorID = 29294 THEN		// Error that no error text table is available
				(* add axis description to error text *)
				brsstrcpy(ADR(status.error.text.active[internal.tmpErrorCount]),ADR(configuration.description));
				brsstrcat(ADR(status.error.text.active[internal.tmpErrorCount]), ADR('- Unable to determine error text, axis error text table not found'));
				state := ST_CHECK_ERROR;
			END_IF

		(***************CHECK AND ACKNOWLEDGE ERRORS********************)
		ST_CHECK_ERROR:
			(* reset all fb execute inputs we use *)
			IF internal.MC_Power_0.Error OR NOT command.power THEN
 				internal.MC_Power_0.Enable := 0;
			END_IF

			IF (internal.MC_BR_ReadAxisError_0.Valid) THEN
				IF (internal.MC_BR_ReadAxisError_0.AxisErrorCount + internal.MC_BR_ReadAxisError_0.AxisWarningCount + internal.MC_BR_ReadAxisError_0.FunctionBlockErrorCount = 0) THEN
					status.error.fault 							:= TRUE;
					internal.MC_BR_ReadAxisError_0.Acknowledge  := FALSE;
					internal.tmpErrorCount						:= 0;

					(* COUNT ALL ERROR STRINGS IN ERROR ARRAY *)
					status.error.count := 0;
					FOR internal.i := 0 TO SIZEOF(status.error.text.active)/SIZEOF(status.error.text.active[0])-1 DO
						IF brsstrlen(ADR(status.error.text.active[internal.i])) <> 0 THEN
							status.error.count := status.error.count + 1;
						ELSE
							EXIT;
						END_IF
					END_FOR

					// wait for acknoledge command
					IF command.errorAcknowledge THEN
						command.errorAcknowledge 	:= FALSE;
						status.error.fault 			:= FALSE;
						status.error.text.last 		:= status.error.text.active;		// copy active to last
						internal.TON_error_read_delay.IN	:= FALSE;
						brsmemset(ADR(status.error.text.active),0,SIZEOF(status.error.text.active)-1);	// clear active list
						status.error.count := 0;

						IF internal.batteryState = ST_BAT_ERROR THEN
							internal.batteryState := ST_BAT_WARNING;
						END_IF

						IF (internal.MC_ReadStatus_0.Errorstop) AND (internal.MC_ReadStatus_0.Valid) THEN
							state := ST_ERROR_RESET;
						ELSE
							IF pAxis.nc_obj_inf.nc_obj_typ = 4 OR pAxis.nc_obj_inf.net_if_typ = 129 THEN
								state := ST_WAIT;
							ELSE
								state := ST_ENCODER_ERROR_RESET;
							END_IF
						END_IF
					END_IF

				(* check if a new errornumber or parid is present, then last error is acknowledged *)
				ELSIF internal.MC_BR_ReadAxisError_0.AxisErrorCount + internal.MC_BR_ReadAxisError_0.AxisWarningCount + internal.MC_BR_ReadAxisError_0.FunctionBlockErrorCount <> 0 THEN
					internal.MC_BR_ReadAxisError_0.Acknowledge	:= FALSE;
					internal.tmpErrorCount						:= internal.tmpErrorCount + 1;
					state 										:= ST_ERROR;
				END_IF
			END_IF

		(*****************RESET AXIS STATE ERRORSTOP********************)
		ST_ERROR_RESET:
			internal.MC_Reset_0.Execute 		:= TRUE;

			IF (internal.MC_Reset_0.Done) THEN
				internal.MC_Reset_0.Execute := 0;
				IF pAxis.nc_obj_inf.nc_obj_typ <> 1 OR pAxis.nc_obj_inf.net_if_typ = 129 THEN 	// 1 = Real axis	129 = sdc_type
					state := ST_WAIT;
				ELSE
					state := ST_ENCODER_ERROR_RESET;
				END_IF
			ELSIF (internal.MC_Reset_0.Error) THEN
				internal.MC_Reset_0.Execute := 0;
				state 						:= ST_ERROR;
			END_IF

		(***************** RESETS ABSOLUTE ENCODER ERRORS ONLY ON ENDAT 2.2 ********************)
		ST_ENCODER_ERROR_RESET:

			CASE internal.substate OF
				0:
					internal.MC_BR_ReadParID_0.Execute 	:= FALSE;
					internal.substate 					:= 1;

				1:	// check encoder type

					internal.MC_BR_ReadParID_0(Axis := configuration.axis, Execute := TRUE , ParID := ACP10PAR_ENCOD_TYPE , DataAddress := ADR(internal.encoderType) , DataType := ncPAR_TYP_USINT);

					IF internal.MC_BR_ReadParID_0.Done THEN
						internal.MC_BR_ReadParID_0.Execute 	:= FALSE;
						internal.substate 					:= 5;
					END_IF

					IF internal.MC_BR_ReadParID_0.Error THEN
						internal.MC_BR_ReadParID_0.Execute 	:= FALSE;
						internal.substate 					:= 0;
						state 			  					:= ST_WAIT;
					END_IF

				5:	// check encoder type
					IF internal.encoderType = ncENDAT THEN
						internal.substate := 10;
					ELSE
						internal.substate := 0;
						state 			  := ST_WAIT;
					END_IF

				10: // check for encoder alarm bit error

					internal.MC_BR_ReadParID_0(Axis := configuration.axis, Execute := TRUE , ParID := ACP10PAR_ENCOD_STATUS , DataAddress := ADR(internal.encoderStatus) , DataType := ncPAR_TYP_UDINT);

					IF internal.MC_BR_ReadParID_0.Done THEN
						internal.MC_BR_ReadParID_0.Execute 	:= FALSE;
						internal.substate 					:= 20;
					END_IF

					IF internal.MC_BR_ReadParID_0.Error THEN
						internal.MC_BR_ReadParID_0.Execute 	:= FALSE;
						internal.substate 					:= 0;
						state 			  					:= ST_WAIT;
					END_IF

				20:	// reset encoder alarm bit error if existing
					internal.encoderReset	:= 1;

					(* check for encoder alarm bit set (bit 5)and encoder warning bit set (bit 8) *)
					IF internal.encoderStatus.5 AND NOT internal.MC_BR_WriteParID_0.Error THEN
						internal.MC_BR_WriteParID_0(Axis := configuration.axis , Execute := TRUE, ParID := ACP10PAR_ENCOD_CMD, DataAddress := ADR(internal.encoderReset) , DataType := ncPAR_TYP_UDINT);

						IF internal.MC_BR_WriteParID_0.Done THEN
							internal.MC_BR_WriteParID_0.Execute := FALSE;
							internal.encoderReset				:= 0;
							internal.substate 					:= 0;
							state								:= ST_WAIT;
						END_IF

					ELSE
						internal.MC_BR_WriteParID_0.Execute := FALSE;
						internal.encoderReset				:= 0;
						internal.substate 					:= 0;
						state 			  					:= ST_WAIT;
					END_IF

			END_CASE

		(******************** SEQUENCE END *************************)

	END_CASE

(***************************************************************
		FUNCTION Block Calls
***************************************************************)

	(************************** MC_POWER ****************************)
	internal.MC_Power_0.Axis := configuration.axis; (* pointer to axis *)
	internal.MC_Power_0();

	(************************** MC_HOME *****************************)
	internal.MC_Home_0.Axis := configuration.axis;
	internal.MC_Home_0();

	(********************** MC_MOVEABSOLUTE *************************)
	internal.MC_MoveAbsolute_0.Axis := configuration.axis;
	internal.MC_MoveAbsolute_0();

	(********************** MC_MOVEADDITIVE *************************)
	internal.MC_MoveAdditive_0.Axis := configuration.axis;
	internal.MC_MoveAdditive_0();

	(********************** MC_MOVEVELOCITY *************************)
	internal.MC_MoveVelocity_0.Axis := configuration.axis;
	internal.MC_MoveVelocity_0();

	(********************** MC_GEARIN *************************)
	internal.MC_GearIn_0.Master := configuration.masterAxis;
	internal.MC_GearIn_0.Slave  := configuration.axis;
//	internal.MC_GearIn_0();

	(********************** MC_GEAROUT *************************)
	internal.MC_GearOut_0.Slave := configuration.axis;
//	internal.MC_GearOut_0();

	(************************** MC_STOP *****************************)
	internal.MC_Stop_0.Axis := configuration.axis;
	internal.MC_Stop_0();

	(************************* MC_BR_INITMODPOS *********************)
	internal.MC_BR_InitModPos_0.Axis := configuration.axis;
	internal.MC_BR_InitModPos_0();

	(************************** MC_HALT *****************************)
	internal.MC_Halt_0.Axis := configuration.axis;
	internal.MC_Halt_0();

	(************************** OTHER *****************************)
	internal.MC_BR_ReadParID_0();
	internal.MC_BR_WriteParID_0();

	(************************* MC_BR_READAXISERROR ***********************)
	internal.MC_BR_ReadAxisError_0.Axis	  := configuration.axis;
	internal.MC_BR_ReadAxisError_0.Mode   := mcTEXT;
	internal.MC_BR_ReadAxisError_0.Enable := 1;

	internal.MC_BR_ReadAxisError_0.Configuration.Format				:= mcNULL;
	internal.MC_BR_ReadAxisError_0.Configuration.DataAddress		:= ADR(internal.tmpErrorArray[0]);
	internal.MC_BR_ReadAxisError_0.Configuration.DataLength			:= SIZEOF(internal.tmpErrorArray);
	internal.MC_BR_ReadAxisError_0.Configuration.LineLength			:= SIZEOF(internal.tmpErrorArray[0]);

	// default error text object name acp10etxen
	IF brsstrlen(ADR(configuration.errorTextObject)) = 0 THEN
		configuration.errorTextObject	:= 'acp10etxen';
	END_IF

	internal.MC_BR_ReadAxisError_0.Configuration.DataObjectName		:= configuration.errorTextObject;
	internal.MC_BR_ReadAxisError_0();

	IF internal.MC_BR_ReadAxisError_0.ErrorRecord.Number = 39014 AND internal.batteryState = ST_BAT_OK THEN //Low battery warning
		internal.batteryState := ST_BAT_ERROR;
	ELSIF internal.MC_BR_ReadAxisError_0.ErrorRecord.Number = 39024  THEN //Encoder positions lost
		internal.batteryState := ST_BAT_POS_LOST;
	END_IF
	(************************** MC_RESET ****************************)
	internal.MC_Reset_0.Axis := configuration.axis;
	internal.MC_Reset_0();

	(************************ MC_BR_CommandError *********************)
	internal.MC_BR_CommandError_0.Axis 		:= configuration.axis;
	internal.MC_BR_CommandError_0.Command	:= parameter.errorSimulationCommand;
	internal.MC_BR_CommandError_0.Execute	:= command.simulateError;
	internal.MC_BR_CommandError_0();

	IF internal.MC_BR_CommandError_0.Done THEN
		internal.MC_BR_CommandError_0.Execute := command.simulateError := FALSE;
	END_IF

	(****************** MC_BR_AXISERRORCOLLECTOR *********************)
	internal.MC_BR_AxisErrorCollector_0.Axis 	:= configuration.axis;
	internal.MC_BR_AxisErrorCollector_0.Enable	:= 1;
	internal.MC_BR_AxisErrorCollector_0();

	(************************ MC_READSTATUS *************************)
	internal.MC_ReadStatus_0.Enable  := 1;
	internal.MC_ReadStatus_0.Axis 	:= configuration.axis;
	internal.MC_ReadStatus_0();

	(******************** MC_READACTUALPOSITION *********************)
	IF  (pAxis.nc_obj_inf.hardware.acp_typ = 0 OR pAxis.nc_obj_inf.hardware.acp_typ = 2) AND pAxis.nc_obj_inf.nc_obj_typ <> 4 THEN		// Check if it is an ACOPOSmulti power supply. if virtual axis its ok
		internal.MC_ReadActualPosition_0.Enable	:= 0;
	ELSIF NOT internal.MC_ReadActualPosition_0.Error AND state < ST_ERROR THEN
		internal.MC_ReadActualPosition_0.Enable	:= 1;
	ELSE
		internal.MC_ReadActualPosition_0.Enable := status.driveStatus.initialized;
	END_IF

	IF NOT configuration.disablePositionReading THEN
		internal.MC_ReadActualPosition_0.Axis	:= configuration.axis;
		internal.MC_ReadActualPosition_0();
		IF (internal.MC_ReadActualPosition_0.Valid) THEN
			status.actPosition := internal.MC_ReadActualPosition_0.Position;
		ELSIF (internal.MC_ReadActualPosition_0.ErrorID <> 0 AND state < ST_ERROR) THEN
			status.actPosition := 0.0;
			state       	   := ST_ERROR;
		END_IF
	ELSE
		status.actPosition := 0.0;
	END_IF

	(******************* MC_BR_WriteParID  *******************)
	internal.MC_BR_WriteParID_1(Axis := configuration.axis);		// write sw end limit ignore

	(******************* MC_BR_INITAXISSUBJECTPAR *******************)
	internal.MC_BR_InitAxisSubjectPar_0.Axis 	:= configuration.axis;
	internal.MC_BR_InitAxisSubjectPar_0.Subject := ncDIG_IN;
	internal.MC_BR_InitAxisSubjectPar_0();

	(******************** MC_BR_SetHardwareInput *******************)
	internal.MC_BR_SetHardwareInputs_0.Enable		:= pAxis.dig_in.level.neg_hw_end >= ncFORCE OR pAxis.dig_in.level.pos_hw_end >= ncFORCE OR
												 	   pAxis.dig_in.level.reference >= ncFORCE OR pAxis.dig_in.level.trigger1 >= ncFORCE OR pAxis.dig_in.level.trigger2 >= ncFORCE;
	internal.MC_BR_SetHardwareInputs_0.HomeSwitch	:= parameter.hwInput.homeReference.input;
	internal.MC_BR_SetHardwareInputs_0.NegHWSwitch	:= parameter.hwInput.negHwLimit.input;
	internal.MC_BR_SetHardwareInputs_0.PosHWSwitch	:= parameter.hwInput.posHwLimit.input;
	internal.MC_BR_SetHardwareInputs_0.Trigger1		:= parameter.hwInput.trigger1.input;
	internal.MC_BR_SetHardwareInputs_0.Trigger2		:= parameter.hwInput.trigger2.input;
//	internal.MC_BR_SetHardwareInputs_0(Axis := configuration.axis);

	(******************** MC_LIMITLOAD *******************)
//	internal.MC_LimitLoad_0(Axis := configuration.axis);

	(******************** MC_READACTUALVELOCITY *********************)
	IF (pAxis.nc_obj_inf.hardware.acp_typ = 0 OR pAxis.nc_obj_inf.hardware.acp_typ = 2) AND pAxis.nc_obj_inf.nc_obj_typ <> 4 THEN		// Check if it is an ACOPOSmulti power supply. if virtual axis its ok
		internal.MC_ReadActualVelocity_0.Enable	:= 0;
	ELSIF NOT internal.MC_ReadActualVelocity_0.Error AND state < ST_ERROR THEN
		internal.MC_ReadActualVelocity_0.Enable	:= 1;
	ELSE
		internal.MC_ReadActualVelocity_0.Enable	:= status.driveStatus.initialized;
	END_IF

	IF NOT configuration.disableVelocityReading THEN
		internal.MC_ReadActualVelocity_0.Axis := configuration.axis;
		internal.MC_ReadActualVelocity_0();
		IF internal.MC_ReadActualVelocity_0.Valid THEN
			status.actVelocity := internal.MC_ReadActualVelocity_0.Velocity;
		ELSIF (internal.MC_ReadActualVelocity_0.ErrorID <> 0 AND state < ST_ERROR) THEN
			status.actVelocity := 0.0;
			state     		   := ST_ERROR;
		END_IF
	ELSE
		status.actVelocity := 0.0;
	END_IF

	(******************** MC_BR_CYCLICREAD LAGERROR *********************)
	IF (pAxis.nc_obj_inf.hardware.acp_typ = 0 OR pAxis.nc_obj_inf.hardware.acp_typ = 2) AND pAxis.nc_obj_inf.nc_obj_typ <> 4 THEN		// Check if it is an ACOPOSmulti power supply. if virtual axis its ok
		internal.MC_BR_CyclicRead_1.Enable	:= 0;
	ELSIF NOT internal.MC_ReadActualVelocity_0.Error AND state < ST_ERROR THEN
		internal.MC_BR_CyclicRead_1.Enable	:= 1;
	ELSE
		internal.MC_BR_CyclicRead_1.Enable	:= status.driveStatus.initialized;
	END_IF

	IF NOT configuration.disableLagErrorReading THEN
		internal.MC_BR_CyclicRead_1.Mode 		:= mcONE_RECORD;
		internal.MC_BR_CyclicRead_1.ParID		:= ACP10PAR_PCTRL_LAG_ERROR;
		internal.MC_BR_CyclicRead_1.DataAddress	:= ADR(status.actLagError);
		internal.MC_BR_CyclicRead_1.DataType	:= ncPAR_TYP_REAL;
		internal.MC_BR_CyclicRead_1.Axis 		:= configuration.axis;
		internal.MC_BR_CyclicRead_1();

		(* scale lag error to PLCopen units *)
		IF configuration.factor <> 0 THEN
			status.actLagError := status.actLagError / UDINT_TO_REAL(configuration.factor);
		END_IF

		IF (internal.MC_BR_CyclicRead_1.ErrorID <> 0 AND state < ST_ERROR) THEN
			status.actLagError := 0.0;
			state     		   := ST_ERROR;
		END_IF
	ELSE
		status.actLagError := 0.0;
	END_IF

	(******************** MC_READACTUALTORQUE *********************)
	// Check if axis is an inverter and a real axis, then enable read torque function
	IF pAxis.nc_obj_inf.hardware.acp_typ = ncACP_TYP_INV AND pAxis.nc_obj_inf.nc_obj_typ = 1 AND NOT internal.MC_ReadActualTorque_0.Error AND state < ST_ERROR THEN
		internal.MC_ReadActualTorque_0.Enable := status.driveStatus.initialized;
	ELSE
		internal.MC_ReadActualTorque_0.Enable := 0;
	END_IF

	IF NOT configuration.disableTorqueReading THEN
		internal.MC_ReadActualTorque_0.Axis	 := configuration.axis;
		internal.MC_ReadActualTorque_0();
		IF internal.MC_ReadActualTorque_0.Valid THEN
			status.actTorque := internal.MC_ReadActualTorque_0.Torque;
		ELSIF (internal.MC_ReadActualTorque_0.ErrorID <> 0 AND state < ST_ERROR) THEN
			status.actTorque := 0.0;
			state   		 := ST_ERROR;
		END_IF
	ELSE
		status.actTorque := 0.0;
	END_IF

	(* get taskclass cycletime info *)
//	IF internal.RTInfo.cycle_time = 0 THEN
//		internal.RTInfo(enable := TRUE);
//	END_IF
//
	internal.TON_error_read_delay(PT := T#1s);
//
//	(* read and save average motor torque *)
//	IF internal.MC_ReadActualTorque_0.Valid AND status.powerOn THEN
//		(* moving average calculation *)
//		internal.filterTime[0] := 500; 				// [ms]
//		internal.filterTime[1] := 5000; 			// [ms]
//
//		FOR internal.i := 0 TO 1 DO
//			internal.filterBase[internal.i] := internal.filterTime[internal.i] / (UDINT_TO_REAL(internal.RTInfo.cycle_time) / 1000);
//
//			IF internal.filterBase[internal.i] < 1 THEN
//				 internal.filterBase[internal.i] := 1;
//			END_IF
//
//			(* calculate filtered position: filterBase = 1 disables the filter *)
//			internal.calcActualValue[internal.i]	 := internal.calcActualValue_old[internal.i] - (internal.calcActualValue_old[internal.i] / internal.filterBase[internal.i]) + (internal.MC_ReadActualTorque_0.Torque / internal.filterBase[internal.i]);
//			internal.calcActualValue_old[internal.i] := internal.calcActualValue[internal.i];
//		END_FOR
//
//		status.torque.actual := brmceil(internal.calcActualValue[0]*100.0)/100.0;
//
//		IF ABS(internal.calcActualValue[0]) > ABS(status.torque.peak) THEN
//			status.torque.peak := brmceil(internal.calcActualValue[0]*100.0)/100.0;
//		END_IF
//
//		IF ABS(internal.calcActualValue[1]) > ABS(status.torque.continous) THEN
//			status.torque.continous := brmceil(internal.calcActualValue[1]*100.0)/100.0;
//		END_IF
//	ELSE
//		status.torque.actual := 0;
//	END_IF
//
//	(* reset continous and peak torque *)
//	IF command.resetTorqueStatus THEN
//		command.resetTorqueStatus := FALSE;
//		status.torque.continous	  := 0.0;
//		status.torque.peak		  := 0.0;
//	END_IF

//	(* read physical motor info *)
//	internal.MC_BR_ReadParID_1.Execute := pAxis.network.phase = 90;		// ACOPOS bootup done, drive ready
//	IF internal.MC_BR_ReadParID_1.Execute AND NOT internal.MC_BR_ReadParID_1.Done AND pAxis.nc_obj_inf.nc_obj_typ <> 4 AND pAxis.nc_obj_inf.net_if_typ = 1 THEN
//		internal.MC_BR_ReadParID_1(Axis := configuration.axis, ParID := ACP10PAR_MOTOR_TORQ_RATED , DataAddress := ADR(info.hw.motor.torqueRated) , DataType := ncPAR_TYP_REAL);
//		info.hw.motor.torqueRated := brmceil(info.hw.motor.torqueRated*100.0)/100.0;
//	ELSIF NOT internal.MC_BR_ReadParID_1.Execute THEN
//		internal.MC_BR_ReadParID_1(Axis := configuration.axis);
//	END_IF
//
//	internal.MC_BR_ReadParID_2.Execute := pAxis.network.phase = 90;		// ACOPOS bootup done, drive ready
//	IF internal.MC_BR_ReadParID_2.Execute AND NOT internal.MC_BR_ReadParID_2.Done AND pAxis.nc_obj_inf.nc_obj_typ <> 4 AND pAxis.nc_obj_inf.net_if_typ = 1 THEN
//		internal.MC_BR_ReadParID_2(Axis := configuration.axis, ParID := ACP10PAR_MOTOR_TORQ_MAX , DataAddress := ADR(info.hw.motor.torqueMaximum) , DataType := ncPAR_TYP_REAL);
//		info.hw.motor.torqueMaximum := brmceil(info.hw.motor.torqueMaximum*100.0)/100.0;
//	ELSIF NOT internal.MC_BR_ReadParID_2.Execute THEN
//		internal.MC_BR_ReadParID_2(Axis := configuration.axis);
//	END_IF
//
//	internal.MC_BR_ReadParID_3.Execute := pAxis.network.phase = 90;		// ACOPOS bootup done, drive ready
//	IF internal.MC_BR_ReadParID_3.Execute AND NOT internal.MC_BR_ReadParID_3.Done AND pAxis.nc_obj_inf.nc_obj_typ <> 4 AND pAxis.nc_obj_inf.net_if_typ = 1 THEN
//		internal.MC_BR_ReadParID_3(Axis := configuration.axis, ParID := ACP10PAR_MOTOR_ORDERTEXT , DataAddress := ADR(info.hw.motor.model) , DataType := ncPAR_TYP_STR32);
//	ELSIF NOT internal.MC_BR_ReadParID_3.Execute THEN
//		internal.MC_BR_ReadParID_3(Axis := configuration.axis);
//	END_IF

//	(* read drive information *)
//	internal.MC_BR_GetHardwareInfo_0.Axis 		:= configuration.axis;
//	internal.MC_BR_GetHardwareInfo_0.Execute 	:= pAxis.network.phase = 90;	// ACOPOS bootup done, drive ready
//	IF internal.MC_BR_GetHardwareInfo_0.Execute AND NOT internal.MC_BR_GetHardwareInfo_0.Done THEN
//		internal.MC_BR_GetHardwareInfo_0();
//	ELSIF NOT internal.MC_BR_GetHardwareInfo_0.Execute THEN
//		internal.MC_BR_GetHardwareInfo_0();
//	END_IF
//
//	info.hw.drive.model 	:= internal.MC_BR_GetHardwareInfo_0.HardwareInfo.Drive.ModelNumber;
//	info.hw.drive.serial 	:= internal.MC_BR_GetHardwareInfo_0.HardwareInfo.Drive.SerialNumber;
//
//	FOR internal.k := 0 TO SIZEOF(info.hw.drive.card)/SIZEOF(info.hw.drive.card[0])-1 DO
//		info.hw.drive.card[internal.k].model 	:= internal.MC_BR_GetHardwareInfo_0.HardwareInfo.Card[internal.k].ModelNumber;
//		info.hw.drive.card[internal.k].serial 	:= internal.MC_BR_GetHardwareInfo_0.HardwareInfo.Card[internal.k].SerialNumber;
//	END_FOR
//
//	(* Read and calculate temperature *)
//	IF pAxis.nc_obj_inf.nc_obj_typ <> 4 AND pAxis.nc_obj_inf.net_if_typ = 1 AND NOT configuration.disableTemperatureReading THEN
//		internal.MC_BR_CyclicRead_0(Axis := configuration.axis, Enable := status.driveStatus.initialized, Mode := mcONE_RECORD, ParID := ACP10PAR_TEMP_MOTOR, DataAddress := ADR(info.hw.motor.temperature) , DataType := ncPAR_TYP_REAL);
//
//		(* moving average temperature calculation *)
//		internal.filterTimeTemp := 3000; // [ms]
//		internal.filterBaseTemp := internal.filterTimeTemp / (UDINT_TO_REAL(internal.RTInfo.cycle_time) / 1000);
//
//		IF internal.filterBaseTemp < 1 THEN
//			 internal.filterBaseTemp := 1;
//		END_IF
//
//		(* calculate filtered position: filterBase = 1 disables the filter *)
//		internal.calcActualValueTemp	 	:= internal.calcActualValueTemp_old - (internal.calcActualValueTemp_old / internal.filterBaseTemp) + (info.hw.motor.temperature / internal.filterBaseTemp);
//		internal.calcActualValueTemp_old 	:= internal.calcActualValueTemp;
//		info.hw.motor.temperature			:= brmceil(ABS(internal.calcActualValueTemp)*10.0)/10.0;
//	ELSE
//		internal.calcActualValueTemp		:= 0.0;
//		internal.calcActualValueTemp_old	:= 0.0;
//		info.hw.motor.temperature 			:= 0.0;
//	END_IF

	(******************** MC_BR_READDRIVEstatus *********************)
	internal.MC_BR_ReadDriveStatus_0.Enable			:= 1;
	internal.MC_BR_ReadDriveStatus_0.Axis	 		:= configuration.axis;
	internal.MC_BR_ReadDriveStatus_0.AdrDriveStatus	:= ADR(internal.tmpDriveStatus);
	internal.MC_BR_ReadDriveStatus_0();

	IF (internal.MC_BR_ReadDriveStatus_0.ErrorID <> 0 AND state < ST_ERROR) THEN
		state := ST_ERROR;
	END_IF

	(* Handling the Description output *)
	IF configuration.description = '' THEN
		IF pAxis.nc_obj_inf.hardware.acp_id = ncACOPOS_1 THEN
			status.axisDescription := 'ACOPOS';
		ELSIF pAxis.nc_obj_inf.hardware.acp_id = ncACOPOS_2 THEN
			status.axisDescription := 'ACOPOS';
		ELSIF pAxis.nc_obj_inf.hardware.acp_id = ncACOPOSmulti THEN
			status.axisDescription := 'ACOPOSmulti';
		ELSIF pAxis.nc_obj_inf.hardware.acp_id = ncACOPOSmulti_PPS THEN
			status.axisDescription := 'ACOPOSmulti PPS';
		ELSIF pAxis.nc_obj_inf.hardware.acp_id = ncACOPOSmicro THEN
			status.axisDescription := 'ACOPOSmicro';
		ELSIF pAxis.nc_obj_inf.hardware.acp_id = ncACOPOSmulti65 THEN
			status.axisDescription := 'ACOPOSmulti65';
		ELSIF pAxis.nc_obj_inf.hardware.acp_id = ncACOPOS_SDC THEN
			status.axisDescription := 'ACOPOS SDC';
		ELSIF pAxis.nc_obj_inf.hardware.acp_id = ncACOPOS_SIM THEN
			status.axisDescription := 'ACOPOS Simulation';
		END_IF

		// Add description if the axis is a virtual axis
		IF pAxis.nc_obj_inf.nc_obj_typ = 4 THEN
			internal.string2 := ' virtual';
			brsstrcat(ADR(status.axisDescription), ADR(internal.string2));(*put second string to end of first one*)
		END_IF

	ELSE
		status.axisDescription := configuration.description;
	END_IF

	(* show the startup phase status *)
	IF pAxis.network.phase = 0 THEN
		info.startupPhase := '0: Communication to ACOPOS is not active';
	ELSIF pAxis.network.phase = 1 THEN
		info.startupPhase := '1: Network initialization was started for unit ACOPOS';
	ELSIF pAxis.network.phase = 5 THEN
		info.startupPhase := '5: Wait for completion of network initialization of NC software with higher startup priority';
	ELSIF pAxis.network.phase = 9 THEN
		info.startupPhase := '9: Wait for communication with ACOPOS BsLoader';
	ELSIF pAxis.network.phase = 10 THEN
		info.startupPhase := '10: Communication with ACOPOS BsLoader has been set up';
	ELSIF pAxis.network.phase = 20 THEN
		info.startupPhase := '20: ACOPOS executes start of BsLoader after SW Reset';
	ELSIF pAxis.network.phase = 30 THEN
		info.startupPhase := '30: Download of BsLoader to unit ACOPOS is executed';
	ELSIF pAxis.network.phase = 31 THEN
		info.startupPhase := '31: Download of BsLoader to other ACOPOS modules is executed';
	ELSIF pAxis.network.phase = 40 THEN
		info.startupPhase := '40: Download of operating system to unit ACOPOS is executed';
	ELSIF pAxis.network.phase = 41 THEN
		info.startupPhase := '41: Download of operating system to other ACOPOS modules is executed';
	ELSIF pAxis.network.phase = 50 THEN
		info.startupPhase := '50: ACOPOS executes start of operating system';
	ELSIF pAxis.network.phase = 55 THEN
		info.startupPhase := '55: Wait for completion of network initialization of NC software with lower startup priority';
	ELSIF pAxis.network.phase = 60 THEN
		info.startupPhase := '60: Default parameters are transferred to the ACOPOS';
	ELSIF pAxis.network.phase = 70 THEN
		info.startupPhase := '70: INIT-ACOPOS parameters are transferred to the ACOPOS';
	ELSIF pAxis.network.phase = 90 THEN
		info.startupPhase := '90: Network initialization complete, drive ready';
	END_IF
(***************** BATTERY STATE MONITOR FOR ACOPOSMICRO WITH ENDAT 2.2 ******************************************)
	IF info.hw.drive.model = '80VD100PD.C000-01' OR
   		info.hw.drive.model = '80VD100PD.C000-14' OR
   		info.hw.drive.model = '80VD100PS.C00X-01' THEN
   		internal.acoposMicroBatMon := TRUE;

		CASE internal.batteryState OF

			ST_BAT_OK:

				status.encoderBatteryStatus.batteryError 	:= FALSE;
				status.encoderBatteryStatus.batteryOK		:= TRUE;
				status.encoderBatteryStatus.batteryWarning	:= FALSE;
				status.encoderBatteryStatus.positionLost  	:= FALSE;

			ST_BAT_ERROR:

				status.encoderBatteryStatus.batteryError 	:= TRUE;
				status.encoderBatteryStatus.batteryOK		:= FALSE;
				status.encoderBatteryStatus.batteryWarning	:= FALSE;
				status.encoderBatteryStatus.positionLost  	:= FALSE;

			ST_BAT_WARNING:

				status.encoderBatteryStatus.batteryError 	:= FALSE;
				status.encoderBatteryStatus.batteryOK		:= FALSE;
				status.encoderBatteryStatus.batteryWarning	:= TRUE;
				status.encoderBatteryStatus.positionLost  	:= FALSE;

				IF command.newBatAcknowledge AND NOT status.powerOn THEN //Reset encoder warning bit - only possible when power is off
					internal.encoderReset := 1;
					internal.MC_BR_WriteParID_0(Axis := configuration.axis , Execute := TRUE, ParID := ACP10PAR_ENCOD_CMD, DataAddress := ADR(internal.encoderReset) , DataType := ncPAR_TYP_UDINT);

					IF internal.MC_BR_WriteParID_0.Done THEN
						internal.MC_BR_WriteParID_0.Execute := FALSE;
						internal.encoderReset				:= 0;
						internal.batteryState				:= ST_BAT_OK;
					END_IF
				END_IF

			ST_BAT_POS_LOST:

				status.encoderBatteryStatus.batteryError 	:= TRUE;
				status.encoderBatteryStatus.batteryOK		:= FALSE;
				status.encoderBatteryStatus.batteryWarning	:= FALSE;
				status.encoderBatteryStatus.positionLost  	:= TRUE;
				IF command.newBatAcknowledge AND NOT status.powerOn THEN //Reset encoder warning bit - only possible when power is off
					internal.encoderReset := 1;
					internal.MC_BR_WriteParID_0(Axis := configuration.axis , Execute := TRUE, ParID := ACP10PAR_ENCOD_CMD, DataAddress := ADR(internal.encoderReset) , DataType := ncPAR_TYP_UDINT);

					IF internal.MC_BR_WriteParID_0.Done THEN
						internal.MC_BR_WriteParID_0.Execute := FALSE;
						internal.encoderReset				:= 0;
						internal.batteryState				:= ST_BAT_OK;
					END_IF
				END_IF

		END_CASE
	ELSE
		internal.batteryState						:= ST_BAT_OK;
		status.encoderBatteryStatus.batteryError 	:= FALSE;
		status.encoderBatteryStatus.batteryOK		:= TRUE;
		status.encoderBatteryStatus.batteryWarning	:= FALSE;
		status.encoderBatteryStatus.positionLost  	:= FALSE;

	END_IF

	(* status *)
	status.stopped 	:= internal.MC_Stop_0.Done;
	status.isHomed 	:= internal.tmpDriveStatus.HomingOk;
	status.powerOn 	:= internal.tmpDriveStatus.ControllerStatus;
	status.inMotion := pAxis.move.mode <> ncOFF AND NOT internal.MC_ReadStatus_0.Disabled AND NOT internal.MC_ReadStatus_0.StandStill;

	(* status drive status *)
	status.driveStatus.controllerReady 		:= internal.tmpDriveStatus.ControllerReady;
	status.driveStatus.driveEnable			:= internal.tmpDriveStatus.DriveEnable;
	status.driveStatus.homeSwitch			:= internal.tmpDriveStatus.HomeSwitch;
	status.driveStatus.negLimitSwitch		:= internal.tmpDriveStatus.NegHWSwitch;
	status.driveStatus.posLimitSwitch		:= internal.tmpDriveStatus.PosHWSwitch;
	status.driveStatus.trigger1				:= internal.tmpDriveStatus.Trigger1;
	status.driveStatus.trigger2				:= internal.tmpDriveStatus.Trigger2;
	status.driveStatus.lagWarning			:= internal.tmpDriveStatus.LagWarning;
	status.driveStatus.initialized			:= internal.tmpDriveStatus.NetworkInit;
	status.driveStatus.simulation			:= internal.tmpDriveStatus.Simulation;

END_FUNCTION_BLOCK
```

#### dstoa.st - Converts an ENUM drive state to ascii
```iecst
(********************************************************************
 * COPYRIGHT -- Bernecker + Rainer
 ********************************************************************
 * Library: BRDK_MC
 * File: dstoa.st
 * Author: olsenm
 * Created: February 20, 2012
 ********************************************************************
 * Implementation of library BRDK_MC
 ********************************************************************)

 (* Converts an ENUM drive state to ascii *)
FUNCTION dstoa

	IF pString <> 0 THEN

		CASE driveState OF

			DISABLED: brsstrcpy(pString, ADR('DISABLED'));

			STANDSTILL: brsstrcpy(pString, ADR('STANDSTILL'));

			HOMING: brsstrcpy(pString, ADR('HOMING'));

			CONTINOUS_MOTION: brsstrcpy(pString, ADR('CONTINOUS_MOTION'));

			DISCRETE_MOTION: brsstrcpy(pString, ADR('DISCRETE_MOTION'));

			SYNCHRONIZED_MOTION: brsstrcpy(pString, ADR('SYNCHRONIZED_MOTION'));

			STOPPING: brsstrcpy(pString, ADR('STOPPING'));

			ERROR_STOP: brsstrcpy(pString, ADR('ERROR_STOP'));

		END_CASE

		dstoa := 1;

	ELSE
		dstoa := 0;
	END_IF

END_FUNCTION
```

- CHANGELOG - brdkMC change log (not shown)

- LICENSE - brdkMC license (not shown)

### Library Logical/Libraries/brdkMU (ANSIC, version 4.04.0) - BRDK machine unit library. Provides functionality to control machines.
Depends on: AsSem, sys_lib, brsystem, brdkSTR

#### brdkEM.typ - brdkEM data types.
```iecst
TYPE
	brdk_em_states_typ :
		( (*Module states. Based on ISA–TR88.00.02 state model.*)
		STATE_DEACTIVATED := 0, (*State Type: Wait
The module has not been activated yet. An activate command will cause an exit from
DEACTIVATED to a ACTIVATING state.*)
		STATE_CLEARING := 1, (*State Type: Acting
Initiated by a state command to clear faults that may have occurred
when ABORTING, and are present in the ABORTED state before
proceeding to a STOPPED state.*)
		STATE_STOPPED := 2, (*State Type: Wait
The machine is powered and stationary after completing the
STOPPING state. All communications with other systems are
functioning (if applicable). A Reset command will cause an exit from
STOPPED to the RESETTING state.*)
		STATE_STARTING := 3, (*State Type: Acting
This state provides the steps needed to start the machine and is a
result of a starting type command (local or remote). Following this
command the machine will begin to Execute.*)
		STATE_IDLE := 4, (*State Type: Wait
This is a state which indicates that RESETTING is complete. This
state maintains the machine conditions which were achieved during
the RESETTING state, and performs operations required when the
machine is in IDLE.*)
		STATE_SUSPENDED := 5, (*State Type: Wait
The machine may be running at a relevant set point speed, but
there is no product being produced while the machine is waiting for
external process conditions to return to normal. When the offending
process conditions return to normal, the SUSPENDED state will
transition to UNSUSPENDING and hence continue towards the
normal EXECUTE state.*)
		STATE_EXECUTE := 6, (*State Type: Dual
Once the machine is processing materials it is deemed to be
executing or in the EXECUTE state. Different machine modes will
result in specific types of EXECUTE activities. For example, if the
machine is in the Production mode, the EXECUTE will result in
products being produced, while in Clean Out mode the EXECUTE
state refers to the action of cleaning the machine.*)
		STATE_STOPPING := 7, (*State Type: Acting
This state executes the logic which brings the machine to a
controlled stop as reflected by the STOPPED state. Normal
STARTING of the machine can not be initiated unless RESETTING
had taken place.*)
		STATE_ABORTING := 8, (*State Type: Acting
The ABORTED state can be entered at any time in response to the
Abort command or on the occurrence of a machine fault. The
aborting logic will bring the machine to a rapid safe stop. Operation
of the emergency stop will cause the machine to be tripped by its
safety system. It will also provide a signal to initiate the
ABORTING State.*)
		STATE_ABORTED := 9, (*State Type: Wait
This state maintains machine status information relevant to the
Abort condition. The machine can only exit the ABORTED state
after an explicit Clear command, subsequently to manual
intervention to correct and reset the detected machine faults.*)
		STATE_HOLDING := 10, (*State Type: Acting
When the machine is in the EXECUTE state, the Hold command
can be used to start HOLDING logic which brings the machine to a
controlled stop or to a state which represents HELD for the
particular unit control mode. A machine can go into this state either
when an internal equipment fault is automatically detected or by an
operator command. The Hold command offers the operator a safe
way to intervene manually in the process (such as removing a
broken bottle from the in-feed) and restarting execution when
conditions are safe. To be able to restart production correctly after
the HELD state, all relevant process set-points and return status of
the procedures at the time of receiving the Hold command must be
saved in the machine controller when executing the HOLDING
procedure.*)
		STATE_HELD := 11, (*State Type: Wait
The HELD state holds the machine's operation while material
blockages are cleared, or to stop throughput while a downstream
problem is resolved, or enable the safe correction of an equipment
fault before the production may be resumed.*)
		STATE_UNHOLDING := 12, (*State Type: Acting
The UNHOLDING state is a response to an Operator command to
resume the EXECUTE state. Issuing the Unhold command will
retrieve the saved set-points and return the status conditions to
prepare the machine to re-enter the normal EXECUTE state.*)
		STATE_SUSPENDING := 13, (*State Type: Acting
This state is a result of a change in monitored conditions due to
process conditions or factors. The trigger event will cause a
temporary suspension of the EXECUTE state. SUSPENDING is
typically the result of starvation of upstream material in-feeds (i.e.,
container feed, beverage feed, crown feed, lubricant feed, etc.) that
is outside the dynamic speed control range or a downstream outfeed
blockage that prevents the machine from EXECUTING
continued steady production. During the controlled sequence of
SUSPENDING the machine will transition to a SUSPENDED state.
The SUSPENDING state might be forced by the operator.*)
		STATE_UNSUSPENDING := 14, (*State Type: Acting
This state is a result of a machine generated request from
SUSPENDED state to go back to the EXECUTE state. The actions
of this state may include ramping up speeds, turning on vacuums,
and the re-engagement of clutches. This state is done prior to
EXECUTE state, and prepares the machine for the EXECUTE state.*)
		STATE_RESETTING := 15, (*State Type: Acting
This state is the result of a RESET command from the STOPPED or
complete state. RESETTING will typically cause a machine to
sound a horn and place the machine in a state where components
are energized awaiting a START command.*)
		STATE_COMPLETING := 16, (*State Type: Acting
This state is an automatic response from the EXECUTE state.
Normal operation has run to completion (i.e., processing of material
at the infeed will stop).*)
		STATE_COMPLETE := 17, (*State Type: Wait
The machine has finished the COMPLETING state and is now
waiting for a Reset command before transitioning to the
RESETTING state.*)
		STATE_DEACTIVATING := 18, (*State Type: Acting
This state is the result of a disabled ACTIVATE command.*)
		STATE_ACTIVATING := 19 (*State Type: Acting
State between DEACTIVATED and STOPPED. This state is done prior to
STOPPED state, and prepares the machine for the STOPPED state.*)
		) := STATE_DEACTIVATED;
	brdk_em_activation_typ :
		( (*Type of activation of equipment module.*)
		BRDK_EM_ACTIVATE := 0, (*Activates the equipment module.*)
		BRDK_EM_DEACTIVATE := 1, (*Deactivated the equipment module.*)
		BRDK_EM_ACTIVATE_BY_PARENT := 2, (*Automatically follows it's parent activation.*)
		BRDK_EM_ACTIVATE_BY_CHILD := 3 (*Activates automatically if a child demand the activation.*)
		) := BRDK_EM_DEACTIVATE;
	brdk_em_command_typ : 	STRUCT  (*Equipment module commands. Based on ISATR88.00.02.*)
		abort : BOOL := FALSE; (*Abort --> Go to STATE_ABORTING - Can be set in all states.*)
		clear : BOOL := FALSE; (*Clear --> Go to STATE_STOPPING - Can only be set in STATE_ABORTED.*)
		stop : BOOL := FALSE; (*Stop --> Go to STATE_STOPPING - Can be set in all states.*)
		reset : BOOL := FALSE; (*Reset --> Go to STATE_RESETTING - Can only be set in STATE_STOPPED.*)
		start : BOOL := FALSE; (*Start --> Go to STATE_STARTING - Can only be set in STATE_IDLE, STATE_SUSPENDED, STATE_HELD.*)
		hold : BOOL := FALSE; (*Hold --> Go to STATE_HOLDING - Can only be set in STATE_EXECUTE.*)
		suspend : BOOL := FALSE; (*Suspend --> Go to STATE_SUSPENDING - Can only be set in STATE_EXECUTE.*)
		complete : BOOL := FALSE; (*Complete --> Go to STATE_COMPLETING - Can only be set in STATE_EXECUTE.*)
		sc : BOOL := FALSE; (*The State Complete indication within the Acting state procedure will cause a state transition to occur. Same functionality as subsuate = SC.*)
	END_STRUCT;
	brdk_em_setup_typ : 	STRUCT  (*Equipment module setup structure.*)
		name : STRING[BRDK_MU_NAME_STRING_SIZE]; (*Name of the module. If empty the name of the task will be given.*)
		nameIdx : DINT := -1; (*Index to be added to name. If -1 no index will be set.*)
		reactTo : brdk_em_setup_react_typ := BRDK_EM_REACT_TO_ALL; (*Indicates which parent state the module should react to.*)
		parent : brdk_mu_setup_module_typ; (*Parameters to setup a parent module.*)
		skipStopSC : BOOL := FALSE; (*When this parameter is set the module will stop even though is not in sub state SC.*)
		sibling : ARRAY[0..BRDK_MU_MAX_SIBLINGS]OF brdk_mu_setup_module_typ; (*List of siblings to a module.*)
		activation : brdk_em_activation_typ := BRDK_EM_ACTIVATE; (*Type of activation of equipment module.*)
		useSubstateSC : BOOL := FALSE; (*Enables the if substate is set to SC it will work as cmd.sc.*)
		lastActivated : BOOL := TRUE; (*Enables the logging.*)
		restore : brdk_em_setup_restore_typ; (*Functionality to restore a module to it's state after a e.g. power failure.*)
	END_STRUCT;
	brdk_em_setup_react_typ :
		( (*Indicates witch command/state the module should react to.*)
		BRDK_EM_REACT_TO_ALL := 0, (*Reacts to all states.*)
		BRDK_EM_REACT_TO_ABORT_AND_STOP := 1, (*Reacts only to abort and stop states.*)
		BRDK_EM_REACT_TO_ABORT_ONLY := 2, (*Reacts only to abort state.*)
		BRDK_EM_REACT_TO_STOP_ONLY := 3, (*Reacts only to stop state.*)
		BRDK_EM_REACT_TO_NONE := 4, (*Doesn't react to any state or mode change. Runs total independent. Equal to the old cmd.ignore.*)
		BRDK_EM_LISTEN_TO_ABORT_AND_STOP := 5, (*The module listen to it's parent aborting and stopping only. Parent don't react to the module.*)
		BRDK_EM_LISTEN_TO_ABORT_ONLY := 6, (*The module listen to it's parent aborting only. Parent don't react to the module.*)
		BRDK_EM_LISTEN_TO_STOP_ONLY := 7 (*The module listen to it's parent stopping only. Parent don't react to the module.*)
		) := BRDK_EM_REACT_TO_ALL;
	brdk_em_setup_restore_typ : 	STRUCT  (*Functionality to restore a module to it's state after a e.g. power failure.*)
		pRestoreStruct : REFERENCE TO brdk_em_restore_module_typ; (*Pointer to the restore structure. Must be defined directly in the task in order to make it retain/permanent.*)
		activate : BOOL := FALSE; (*Activates the storing of the module information in the restore structure. This is to avoid overwriting the restore information.*)
	END_STRUCT;
	brdk_em_status_typ : 	STRUCT  (*Equipment module status.*)
		state : STRING[21]; (*String representation of the state.*)
		substate : STRING[BRDK_MU_MAX_DESCRIPTION_STRING]; (*Can be set in the task to descripe what the module is doing in this substate.*)
		mode : STRING[21]; (*String representation of the mode.*)
		name : STRING[BRDK_MU_NAME_STRING_SIZE]; (*Name of the module. If empty the name of the task will be given.*)
		time : UDINT; (*[ms] Actual time spend in the current state.*)
		last : ARRAY[0..BRDK_MU_MAX_LAST_SIZE]OF STRING[43]; (*The last state and substate the module was in and the spend time.*)
		childCount : UDINT; (*How many children are registered.*)
		waitingFor : brdk_em_waiting_for_typ; (*Info: Which child the parent and the underlying modules are waiting for.*)
		interruptedBy : brdk_em_interrupted_by_typ; (*Info: Which child interruped the parent by going into STOPPING or ABORTING.*)
		color : brdk_em_color_typ; (*Color depending af the unit state.*)
		lightTree : brdk_em_status_light_tree_typ; (*Light tree indicating the status of the module.*)
		cycleTime : UDINT; (*[µsec] Cycle time of the modules's task.*)
		parent : brdk_mu_status_module_typ; (*Information about the parent.*)
		sibling : ARRAY[0..BRDK_MU_MAX_SIBLINGS]OF brdk_mu_status_module_typ; (*List of available siblings.*)
		unvalidatedCmd : BOOL; (*Indicates that the current state cannot accept the given command.*)
		unvalidatedMode : BOOL; (*Indicates that the current state cannot accept the given mode change. Modes can only be changed in STATE_STOPPED and in STATE_ACTIVATING. The status flag will be reset by a state change.*)
		sleeping : BOOL; (*Indicates that the module is sleeping meaning that the module is not being executed because a new instance is being transferred.*)
		level : UDINT; (*Level in the hierarchy. Parent is level 0.*)
	END_STRUCT;
	brdk_em_status_light_tree_typ : 	STRUCT  (*Light tree indicating the status of the module. The idea of the light tree status is that it can be mapped directly to an output module.*)
		red : BOOL := FALSE; (*Color red.*)
		yellow : BOOL := FALSE; (*Color yellow.*)
		blue : BOOL := FALSE; (*Color blue.*)
		green : BOOL := FALSE; (*Color green.*)
	END_STRUCT;
	brdk_em_color_typ :
		( (*Color to display the current state.*)
		GREY := 0, (*Wait State - Unit is disabled*)
		BLUE := 1, (*Wait State – A stable state used to identify that a Unit has achieved a defined set of
conditions. In such a state the Unit is holding or maintaining a status until transitioning
to an Acting state (White color). The unit is powered and stationary.*)
		WHITE := 2, (*Acting State – A state which represents some processing activity, for example ramping
up speed.
It implies the single or repeated execution of processing steps in a logical order, for a
finite time or until a specific condition has been reached, for example within the
Starting state the quality of the received data is checking, before raping up speed for
execution.*)
		GREEN := 3, (*Dual State - The Unit is in a stable acting state. The unit is running and drives are active
and the unit is producing.*)
		RED := 4, (*Wait state – A state which represents an error state on the Unit. In this state the Unit is
not producing, until the operator have managed to make a transition to the EXECUTING
state. The state holds the units operation in a safe environment, until the command
unhold are executed. For example a material blockage will move the unit into the HELD
state. The unit will leave the state HELD, when the operator have entered the unit,
removed the the bloackage, and enabled all safeguards and activated the Unhold
command.*)
		ORANGE := 5 (*Wait State – A state which represents an error state on the line and the Unit is running
at a relevant set point speed, but there is no product being produced while the unit is
waiting for external process conditions to return to normal. The unit will also enter this
state if the operator want to have a break.*)
		) := GREY;
	brdk_em_interrupted_by_typ : 	STRUCT  (*Tells which unit has interrupted the hierarchy into STATE_ABORTING or STATE_STOPPING.*)
		name : STRING[BRDK_MU_NAME_STRING_SIZE]; (*Name of the child that has interrupted the parent.*)
		state : brdk_em_states_typ := STATE_DEACTIVATED; (*State info.*)
		substate : UINT := 0; (*Substate info.*)
	END_STRUCT;
	brdk_em_waiting_for_typ : 	STRUCT  (*Tells which child module the hierarchy are waiting for. Can be that the modules are waiting for more children, but only one of them a shown at a time.*)
		name : STRING[BRDK_MU_NAME_STRING_SIZE]; (*Name of the child that the parent is waiting for.*)
		substate : STRING[BRDK_MU_MAX_DESCRIPTION_STRING]; (*Child substate.*)
	END_STRUCT;
	brdk_em_internal_typ : 	STRUCT  (*Internal variables.*)
		SemCreate_0 : SemCreate; (*Module semaphore.*)
		old : brdk_em_state_old_typ; (*Last state info.*)
		flashTime : UDINT := 0; (*Flash time counter.*)
		initSubstate : UINT := 0; (*Internal temp sub state to be used in STATE_DEACTIVATED.*)
		pInterrupter : UDINT := 0; (*Pointer to the module that interrupted.*)
		findParent : BOOL := FALSE; (*The module automatically finds it's parent's state.*)
		muList : brdk_em_internal_mu_list_typ; (*Holds index's in the MU list.*)
		cmdSC : BOOL; (*Internal command state complete.*)
	END_STRUCT;
	brdk_em_state_old_typ : 	STRUCT  (*Holds the old states.*)
		state : brdk_em_states_typ := STATE_DEACTIVATED; (*Old state.*)
		substate : UINT := 0; (*Old substate.*)
		mode : DINT := 0; (*Old mode.*)
		reactTo : brdk_em_setup_react_typ := BRDK_EM_REACT_TO_ALL; (*Old reactTo.*)
	END_STRUCT;
	brdk_em_internal_mu_list_typ : 	STRUCT  (*Holds index's in the MU list.*)
		idx : DINT := -1; (*Own index in the mu list.*)
		parentIdx : DINT := -1; (*Parent index in the mu list.*)
		siblingIdx : ARRAY[0..BRDK_MU_MAX_SIBLINGS]OF DINT := [4(-1)]; (*Siblings index in the mu list.*)
		childrenIdx : ARRAY[0..BRDK_EM_MAX_CHILDREN]OF DINT; (*Children index in the mu list.*)
	END_STRUCT;
	brdk_em_restore_module_typ : 	STRUCT  (*Hold information that can be used to restore to it's active state in the case of a power failure.*)
		state : brdk_em_states_typ; (*Restored state.*)
		substate : UINT; (*Restored sub state.*)
		sc : BOOL; (*Restores state complete.*)
		mode : UINT; (*Restore mode.*)
	END_STRUCT;
END_TYPE
```

#### brdkCM.typ - brdkCM data types.
```iecst
TYPE
	brdk_cm_setup_typ : 	STRUCT  (*Equipment module setup structure.*)
		name : STRING[BRDK_MU_NAME_STRING_SIZE]; (*Name of the module.*)
		nameIdx : DINT := -1; (*Index to be added to name. If -1 no index will be set.*)
		parent : brdk_mu_setup_module_typ; (*Parameters to setup a parent module.*)
		sibling : ARRAY[0..BRDK_MU_MAX_SIBLINGS]OF brdk_mu_setup_module_typ; (*List of siblings to a module.*)
		lastActivated : BOOL := TRUE; (*Enables the logging of the last state and sub state.*)
	END_STRUCT;
	brdk_cm_status_typ : 	STRUCT  (*Control module status type.*)
		ready : BOOL := FALSE; (*Control module is ready for use.*)
		state : STRING[BRDK_MU_MAX_DESCRIPTION_STRING]; (*Can be set in the task to descripe what the module is doing in this state.*)
		time : UDINT; (*[ms] Actual time spend in the current state.*)
		last : ARRAY[0..BRDK_MU_MAX_LAST_SIZE]OF STRING[25]; (*The last state the module was in.*)
		cycleTime : UDINT; (*[µsec] Cycle time of the modules's task.*)
		parent : brdk_mu_status_module_typ; (*Information about the parent.*)
		sibling : ARRAY[0..BRDK_MU_MAX_SIBLINGS]OF brdk_mu_status_module_typ; (*List of available siblings.*)
		sleeping : BOOL; (*Indicates that the module is sleeping meaning that the module is not being executed because a new instance is being transferred.*)
		level : UDINT; (*Level in the hierarchy. Parent is level 0.*)
		name : STRING[BRDK_MU_NAME_STRING_SIZE]; (*Name of the module.*)
	END_STRUCT;
	brdk_cm_internal_mu_list_typ : 	STRUCT  (*Holds index's in the MU list.*)
		idx : DINT := -1; (*Own index in the mu list.*)
		parentIdx : DINT := -1; (*Parent index in the mu list.*)
		siblingIdx : ARRAY[0..BRDK_MU_MAX_SIBLINGS]OF DINT := [4(-1)]; (*Siblings index in the mu list.*)
	END_STRUCT;
	brdk_cm_internal_typ : 	STRUCT  (*Control module internal variables.*)
		initSubstate : UINT := 0; (*Internal temp sub state to be used in INIT PROGRAM.*)
		muList : brdk_cm_internal_mu_list_typ; (*Holds index's in the MU list.*)
		old : brdk_cm_state_old_typ; (*Holds the old states.*)
	END_STRUCT;
	brdk_cm_state_old_typ : 	STRUCT  (*Holds the old states.*)
		state : UINT; (*Old CM state.*)
		substate : UINT; (*Old CM substate.*)
	END_STRUCT;
END_TYPE
```
